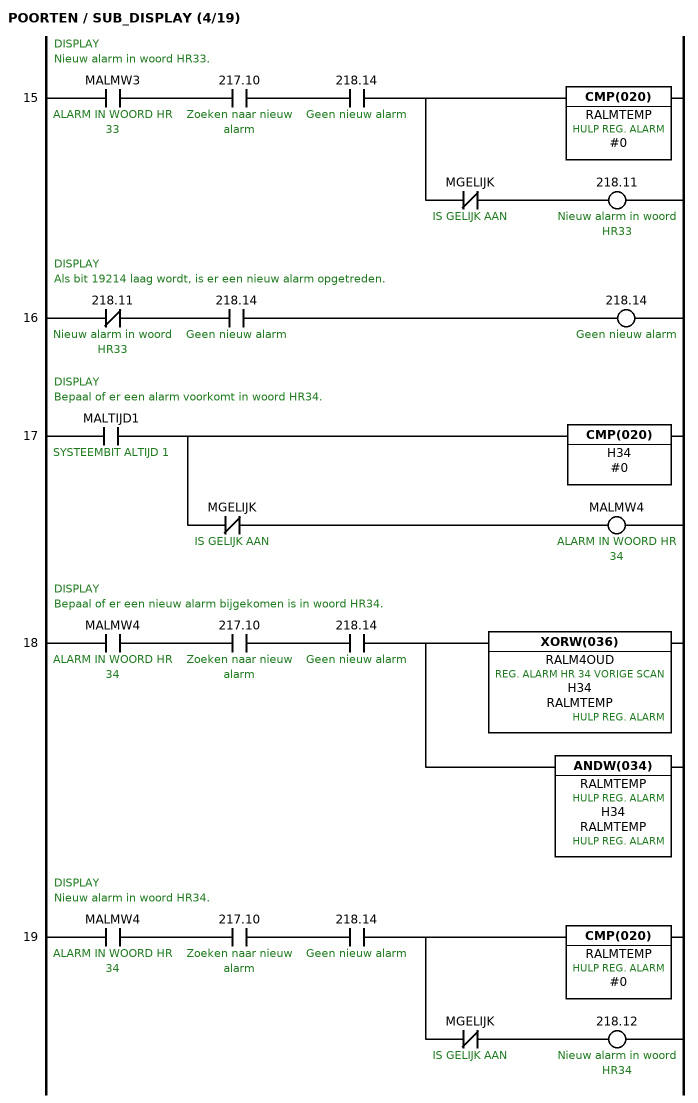
; [picture p469: POORTEN / SUB_DISPLAY, rungs 15-19]
; rung 15: DISPLAY / Nieuw alarm in woord HR33.
LD MALMW3  ; ALARM IN WOORD HR 33
AND 217.10  ; Zoeken naar nieuw alarm
AND 218.14  ; Geen nieuw alarm
CMP(020) RALMTEMP #0  ; HULP REG. ALARM
ANDNOT MGELIJK  ; IS GELIJK AAN
OUT 218.11  ; Nieuw alarm in woord HR33
; rung 16: DISPLAY / Als bit 19214 laag wordt, is er een nieuw alarm opgetreden.
LDNOT 218.11  ; Nieuw alarm in woord HR33
AND 218.14  ; Geen nieuw alarm
OUT 218.14  ; Geen nieuw alarm
; rung 17: DISPLAY / Bepaal of er een alarm voorkomt in woord HR34.
LD MALTIJD1  ; SYSTEEMBIT ALTIJD 1
CMP(020) H34 #0
ANDNOT MGELIJK  ; IS GELIJK AAN
OUT MALMW4  ; ALARM IN WOORD HR 34
; rung 18: DISPLAY / Bepaal of er een nieuw alarm bijgekomen is in woord HR34.
LD MALMW4  ; ALARM IN WOORD HR 34
AND 217.10  ; Zoeken naar nieuw alarm
AND 218.14  ; Geen nieuw alarm
XORW(036) RALM4OUD H34 RALMTEMP  ; REG. ALARM HR 34 VORIGE SCAN, HULP REG. ALARM
ANDW(034) RALMTEMP H34 RALMTEMP  ; HULP REG. ALARM
; rung 19: DISPLAY / Nieuw alarm in woord HR34.
LD MALMW4  ; ALARM IN WOORD HR 34
AND 217.10  ; Zoeken naar nieuw alarm
AND 218.14  ; Geen nieuw alarm
CMP(020) RALMTEMP #0  ; HULP REG. ALARM
ANDNOT MGELIJK  ; IS GELIJK AAN
OUT 218.12  ; Nieuw alarm in woord HR34

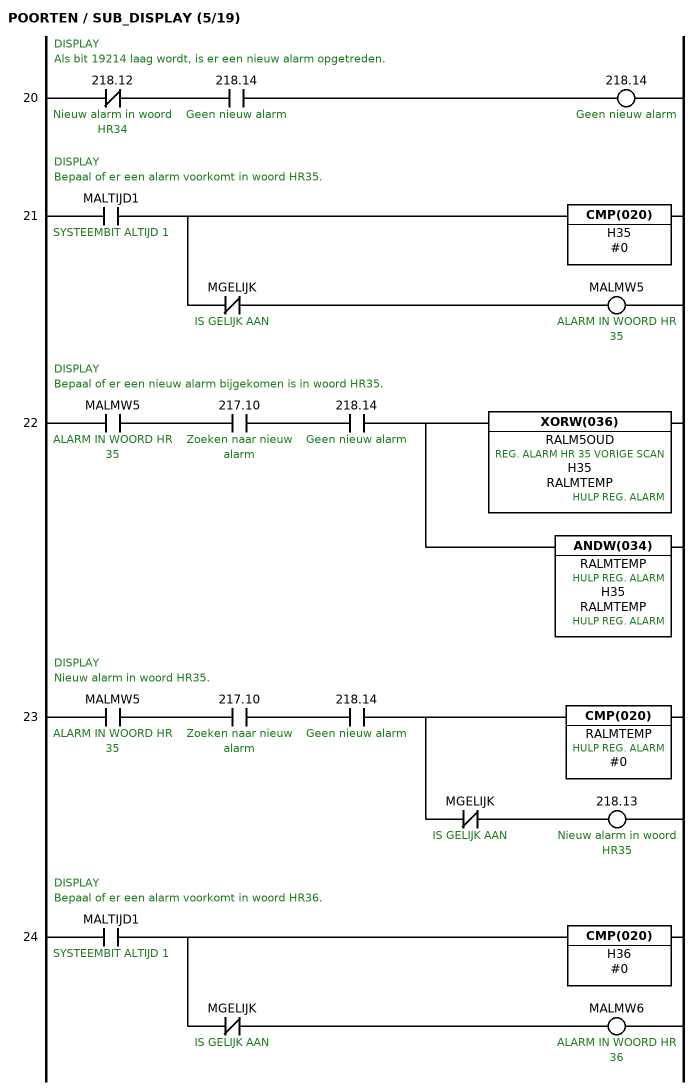
; rung 20: DISPLAY / Als bit 19214 laag wordt, is er een nieuw alarm opgetreden.
LDNOT 218.12  ; Nieuw alarm in woord HR34
AND 218.14  ; Geen nieuw alarm
OUT 218.14  ; Geen nieuw alarm
; rung 21: DISPLAY / Bepaal of er een alarm voorkomt in woord HR35.
LD MALTIJD1  ; SYSTEEMBIT ALTIJD 1
CMP(020) H35 #0
ANDNOT MGELIJK  ; IS GELIJK AAN
OUT MALMW5  ; ALARM IN WOORD HR 35
; rung 22: DISPLAY / Bepaal of er een nieuw alarm bijgekomen is in woord HR35.
LD MALMW5  ; ALARM IN WOORD HR 35
AND 217.10  ; Zoeken naar nieuw alarm
AND 218.14  ; Geen nieuw alarm
XORW(036) RALM5OUD H35 RALMTEMP  ; REG. ALARM HR 35 VORIGE SCAN, HULP REG. ALARM
ANDW(034) RALMTEMP H35 RALMTEMP  ; HULP REG. ALARM
; rung 23: DISPLAY / Nieuw alarm in woord HR35.
LD MALMW5  ; ALARM IN WOORD HR 35
AND 217.10  ; Zoeken naar nieuw alarm
AND 218.14  ; Geen nieuw alarm
CMP(020) RALMTEMP #0  ; HULP REG. ALARM
ANDNOT MGELIJK  ; IS GELIJK AAN
OUT 218.13  ; Nieuw alarm in woord HR35
; rung 24: DISPLAY / Bepaal of er een alarm voorkomt in woord HR36.
LD MALTIJD1  ; SYSTEEMBIT ALTIJD 1
CMP(020) H36 #0
ANDNOT MGELIJK  ; IS GELIJK AAN
OUT MALMW6  ; ALARM IN WOORD HR 36

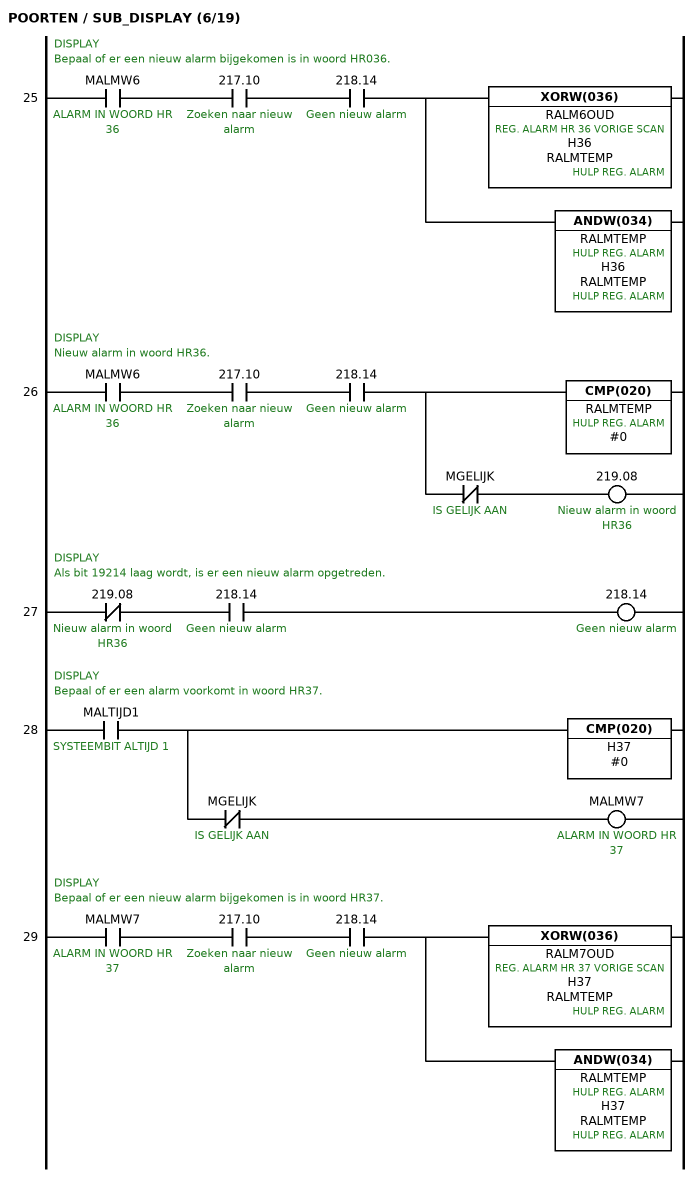
; rung 25: DISPLAY / Bepaal of er een nieuw alarm bijgekomen is in woord HR036.
LD MALMW6  ; ALARM IN WOORD HR 36
AND 217.10  ; Zoeken naar nieuw alarm
AND 218.14  ; Geen nieuw alarm
XORW(036) RALM6OUD H36 RALMTEMP  ; REG. ALARM HR 36 VORIGE SCAN, HULP REG. ALARM
ANDW(034) RALMTEMP H36 RALMTEMP  ; HULP REG. ALARM
; rung 26: DISPLAY / Nieuw alarm in woord HR36.
LD MALMW6  ; ALARM IN WOORD HR 36
AND 217.10  ; Zoeken naar nieuw alarm
AND 218.14  ; Geen nieuw alarm
CMP(020) RALMTEMP #0  ; HULP REG. ALARM
ANDNOT MGELIJK  ; IS GELIJK AAN
OUT 219.08  ; Nieuw alarm in woord HR36
; rung 27: DISPLAY / Als bit 19214 laag wordt, is er een nieuw alarm opgetreden.
LDNOT 219.08  ; Nieuw alarm in woord HR36
AND 218.14  ; Geen nieuw alarm
OUT 218.14  ; Geen nieuw alarm
; rung 28: DISPLAY / Bepaal of er een alarm voorkomt in woord HR37.
LD MALTIJD1  ; SYSTEEMBIT ALTIJD 1
CMP(020) H37 #0
ANDNOT MGELIJK  ; IS GELIJK AAN
OUT MALMW7  ; ALARM IN WOORD HR 37
; rung 29: DISPLAY / Bepaal of er een nieuw alarm bijgekomen is in woord HR37.
LD MALMW7  ; ALARM IN WOORD HR 37
AND 217.10  ; Zoeken naar nieuw alarm
AND 218.14  ; Geen nieuw alarm
XORW(036) RALM7OUD H37 RALMTEMP  ; REG. ALARM HR 37 VORIGE SCAN, HULP REG. ALARM
ANDW(034) RALMTEMP H37 RALMTEMP  ; HULP REG. ALARM

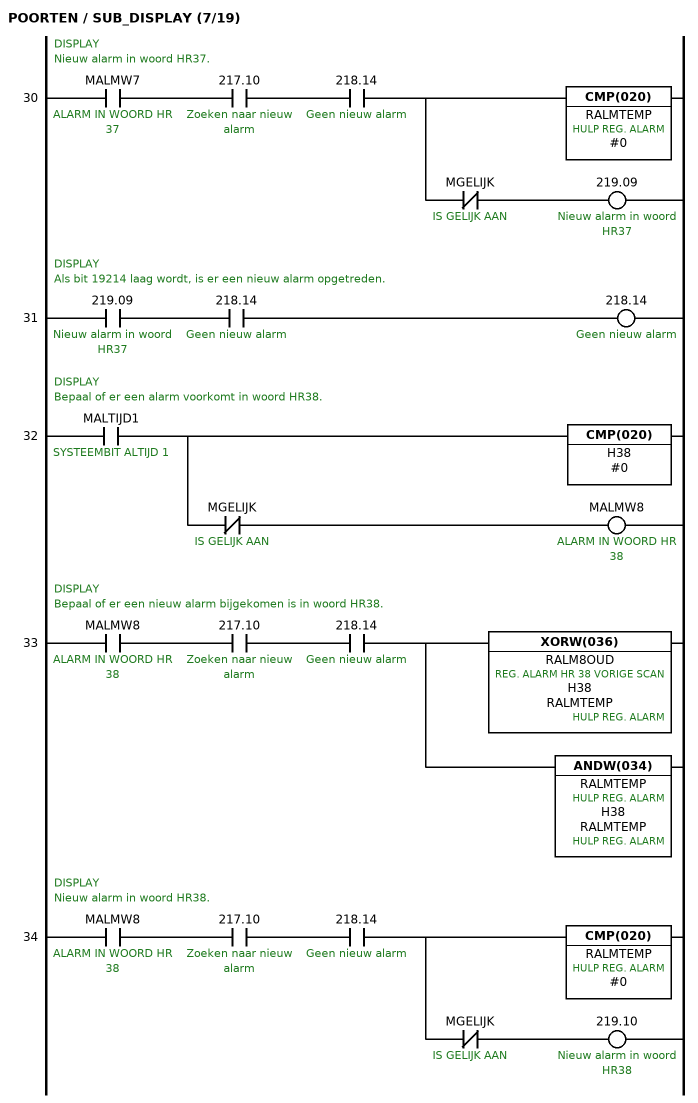
; rung 30: DISPLAY / Nieuw alarm in woord HR37.
LD MALMW7  ; ALARM IN WOORD HR 37
AND 217.10  ; Zoeken naar nieuw alarm
AND 218.14  ; Geen nieuw alarm
CMP(020) RALMTEMP #0  ; HULP REG. ALARM
ANDNOT MGELIJK  ; IS GELIJK AAN
OUT 219.09  ; Nieuw alarm in woord HR37
; rung 31: DISPLAY / Als bit 19214 laag wordt, is er een nieuw alarm opgetreden.
LD 219.09  ; Nieuw alarm in woord HR37
AND 218.14  ; Geen nieuw alarm
OUT 218.14  ; Geen nieuw alarm
; rung 32: DISPLAY / Bepaal of er een alarm voorkomt in woord HR38.
LD MALTIJD1  ; SYSTEEMBIT ALTIJD 1
CMP(020) H38 #0
ANDNOT MGELIJK  ; IS GELIJK AAN
OUT MALMW8  ; ALARM IN WOORD HR 38
; rung 33: DISPLAY / Bepaal of er een nieuw alarm bijgekomen is in woord HR38.
LD MALMW8  ; ALARM IN WOORD HR 38
AND 217.10  ; Zoeken naar nieuw alarm
AND 218.14  ; Geen nieuw alarm
XORW(036) RALM8OUD H38 RALMTEMP  ; REG. ALARM HR 38 VORIGE SCAN, HULP REG. ALARM
ANDW(034) RALMTEMP H38 RALMTEMP  ; HULP REG. ALARM
; rung 34: DISPLAY / Nieuw alarm in woord HR38.
LD MALMW8  ; ALARM IN WOORD HR 38
AND 217.10  ; Zoeken naar nieuw alarm
AND 218.14  ; Geen nieuw alarm
CMP(020) RALMTEMP #0  ; HULP REG. ALARM
ANDNOT MGELIJK  ; IS GELIJK AAN
OUT 219.10  ; Nieuw alarm in woord HR38

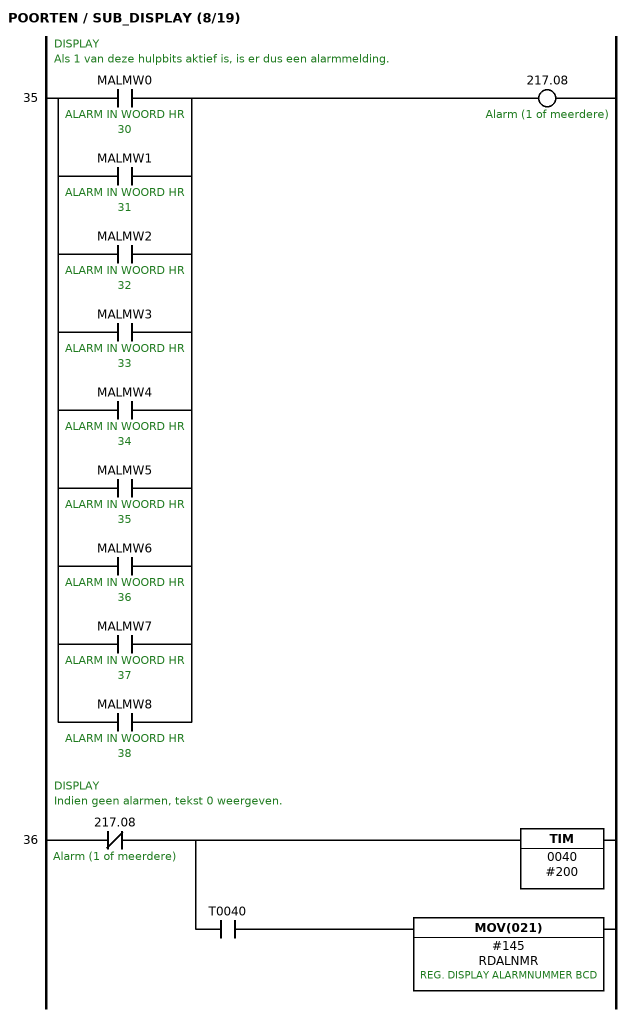
; rung 35: DISPLAY / Als 1 van deze hulpbits aktief is, is er dus een alarmmelding.
LD MALMW0  ; ALARM IN WOORD HR 30
OR MALMW1  ; ALARM IN WOORD HR 31
OR MALMW2  ; ALARM IN WOORD HR 32
OR MALMW3  ; ALARM IN WOORD HR 33
OR MALMW4  ; ALARM IN WOORD HR 34
OR MALMW5  ; ALARM IN WOORD HR 35
OR MALMW6  ; ALARM IN WOORD HR 36
OR MALMW7  ; ALARM IN WOORD HR 37
OR MALMW8  ; ALARM IN WOORD HR 38
OUT 217.08  ; Alarm (1 of meerdere)
; rung 36: DISPLAY / Indien geen alarmen, tekst 0 weergeven.
LDNOT 217.08  ; Alarm (1 of meerdere)
TIM 0040 #200
AND T0040
MOV(021) #145 RDALNMR  ; REG. DISPLAY ALARMNUMMER BCD

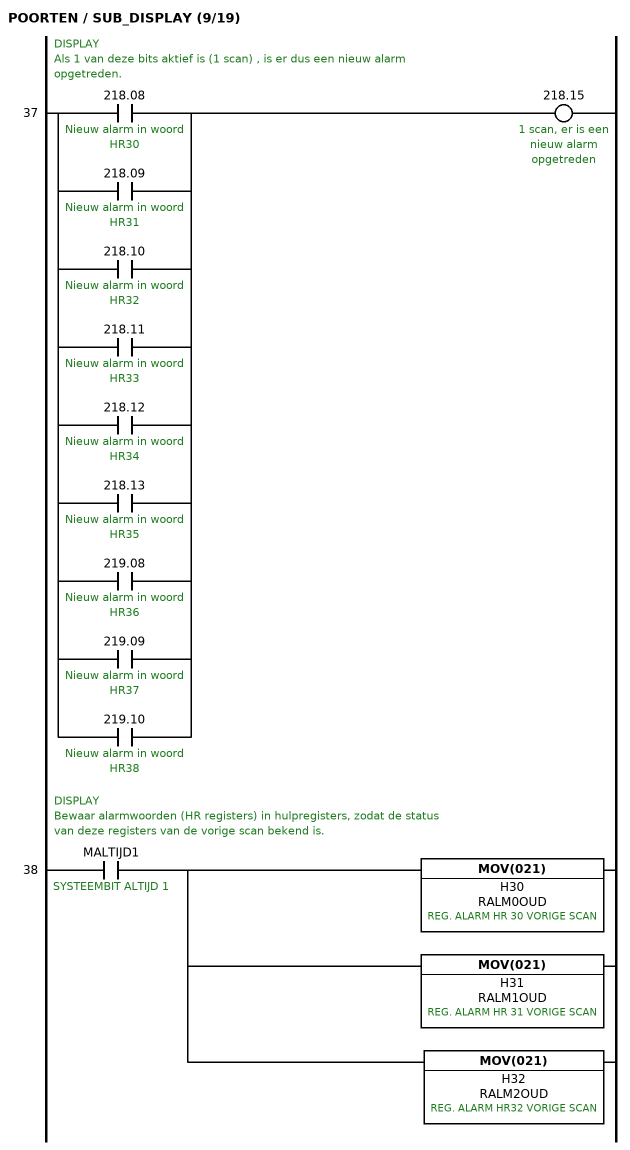
; rung 37: DISPLAY / Als 1 van deze bits aktief is (1 scan) , is er dus een nieuw alarm / opgetreden.
LD 218.08  ; Nieuw alarm in woord HR30
OR 218.09  ; Nieuw alarm in woord HR31
OR 218.10  ; Nieuw alarm in woord HR32
OR 218.11  ; Nieuw alarm in woord HR33
OR 218.12  ; Nieuw alarm in woord HR34
OR 218.13  ; Nieuw alarm in woord HR35
OR 219.08  ; Nieuw alarm in woord HR36
OR 219.09  ; Nieuw alarm in woord HR37
OR 219.10  ; Nieuw alarm in woord HR38
OUT 218.15  ; 1 scan, er is een nieuw alarm opgetreden
; rung 38: DISPLAY / Bewaar alarmwoorden (HR registers) in hulpregisters, zodat de status / van deze registers van de vorige scan bekend is.
LD MALTIJD1  ; SYSTEEMBIT ALTIJD 1
MOV(021) H30 RALM0OUD  ; REG. ALARM HR 30 VORIGE SCAN
MOV(021) H31 RALM1OUD  ; REG. ALARM HR 31 VORIGE SCAN
MOV(021) H32 RALM2OUD  ; REG. ALARM HR32 VORIGE SCAN

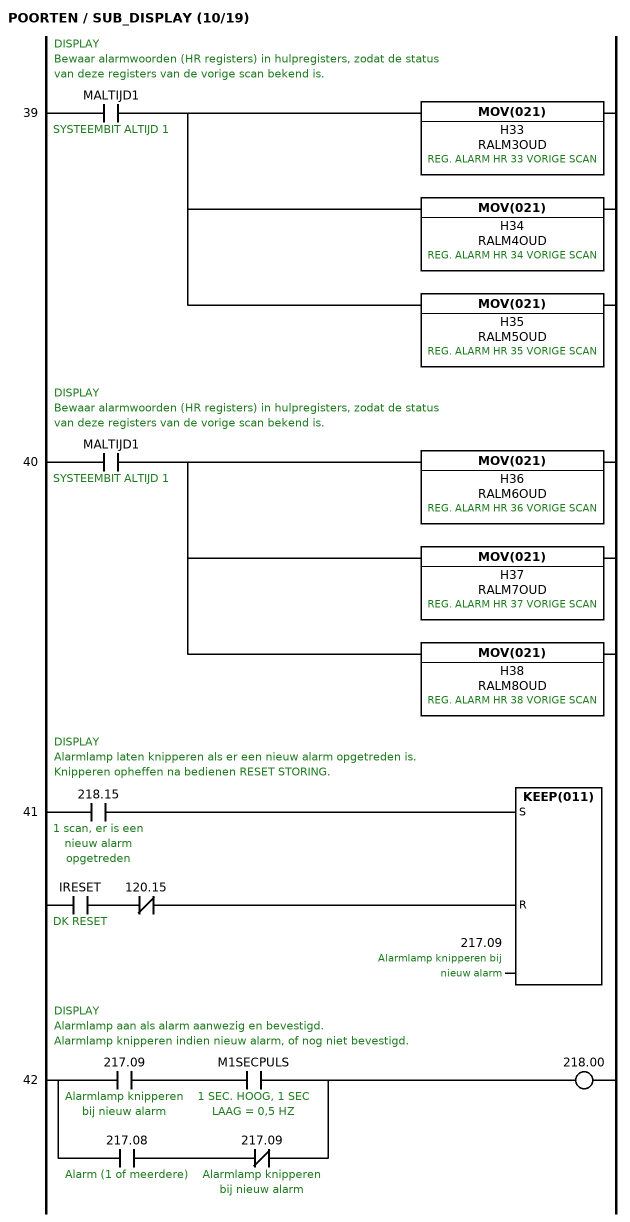
; rung 39: DISPLAY / Bewaar alarmwoorden (HR registers) in hulpregisters, zodat de status / van deze registers van de vorige scan bekend is.
LD MALTIJD1  ; SYSTEEMBIT ALTIJD 1
MOV(021) H33 RALM3OUD  ; REG. ALARM HR 33 VORIGE SCAN
MOV(021) H34 RALM4OUD  ; REG. ALARM HR 34 VORIGE SCAN
MOV(021) H35 RALM5OUD  ; REG. ALARM HR 35 VORIGE SCAN
; rung 40: DISPLAY / Bewaar alarmwoorden (HR registers) in hulpregisters, zodat de status / van deze registers van de vorige scan bekend is.
LD MALTIJD1  ; SYSTEEMBIT ALTIJD 1
MOV(021) H36 RALM6OUD  ; REG. ALARM HR 36 VORIGE SCAN
MOV(021) H37 RALM7OUD  ; REG. ALARM HR 37 VORIGE SCAN
MOV(021) H38 RALM8OUD  ; REG. ALARM HR 38 VORIGE SCAN
; rung 41: DISPLAY / Alarmlamp laten knipperen als er een nieuw alarm opgetreden is. / Knipperen opheffen na bedienen RESET STORING.
LD 218.15  ; 1 scan, er is een nieuw alarm opgetreden
LD IRESET  ; DK RESET
ANDNOT 120.15
KEEP(011) 217.09  ; Alarmlamp knipperen bij nieuw alarm
; rung 42: DISPLAY / Alarmlamp aan als alarm aanwezig en bevestigd. / Alarmlamp knipperen indien nieuw alarm, of nog niet bevestigd.
LD 217.09  ; Alarmlamp knipperen bij nieuw alarm
AND M1SECPULS  ; 1 SEC. HOOG, 1 SEC LAAG = 0,5 HZ
LD 217.08  ; Alarm (1 of meerdere)
ANDNOT 217.09  ; Alarmlamp knipperen bij nieuw alarm
ORLD
OUT 218.00

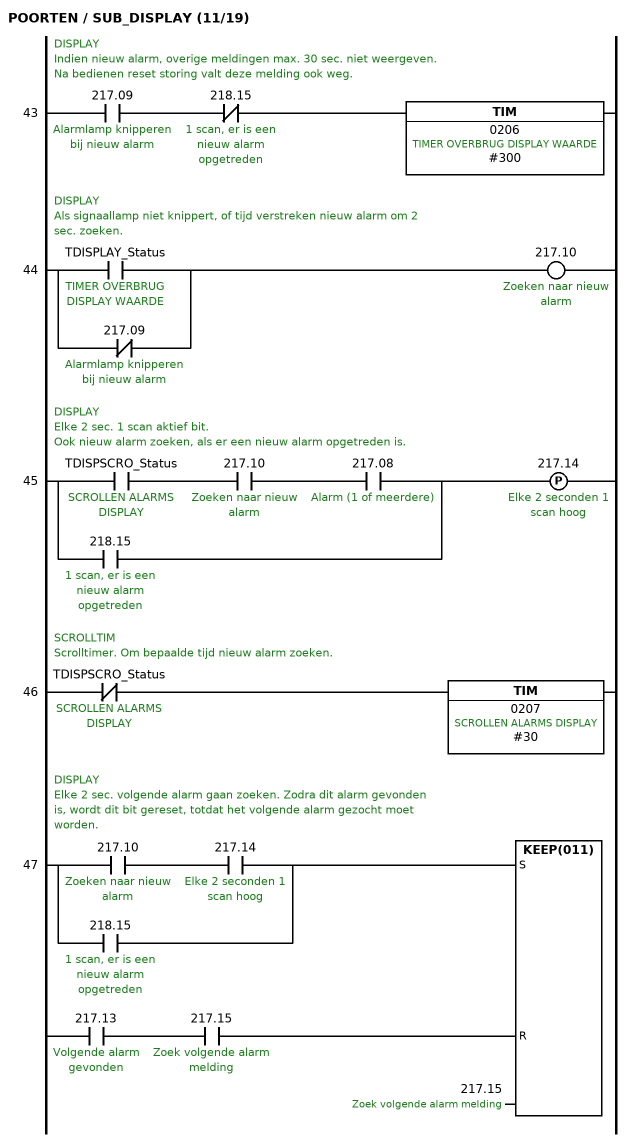
; rung 43: DISPLAY / Indien nieuw alarm, overige meldingen max. 30 sec. niet weergeven. / Na bedienen reset storing valt deze melding ook weg.
LD 217.09  ; Alarmlamp knipperen bij nieuw alarm
ANDNOT 218.15  ; 1 scan, er is een nieuw alarm opgetreden
TIM 0206 #300  ; TIMER OVERBRUG DISPLAY WAARDE
; rung 44: DISPLAY / Als signaallamp niet knippert, of tijd verstreken nieuw alarm om 2 / sec. zoeken.
LD TDISPLAY_Status  ; TIMER OVERBRUG DISPLAY WAARDE
ORNOT 217.09  ; Alarmlamp knipperen bij nieuw alarm
OUT 217.10  ; Zoeken naar nieuw alarm
; rung 45: DISPLAY / Elke 2 sec. 1 scan aktief bit. / Ook nieuw alarm zoeken, als er een nieuw alarm opgetreden is.
LD TDISPSCRO_Status  ; SCROLLEN ALARMS DISPLAY
AND 217.10  ; Zoeken naar nieuw alarm
AND 217.08  ; Alarm (1 of meerdere)
OR 218.15  ; 1 scan, er is een nieuw alarm opgetreden
DIFU(013) 217.14  ; Elke 2 seconden 1 scan hoog
; rung 46: SCROLLTIM / Scrolltimer. Om bepaalde tijd nieuw alarm zoeken.
LDNOT TDISPSCRO_Status  ; SCROLLEN ALARMS DISPLAY
TIM 0207 #30  ; SCROLLEN ALARMS DISPLAY
; rung 47: DISPLAY / Elke 2 sec. volgende alarm gaan zoeken. Zodra dit alarm gevonden / is, wordt dit bit gereset, totdat het volgende alarm gezocht moet / worden.
LD 217.10  ; Zoeken naar nieuw alarm
AND 217.14  ; Elke 2 seconden 1 scan hoog
OR 218.15  ; 1 scan, er is een nieuw alarm opgetreden
LD 217.13  ; Volgende alarm gevonden
AND 217.15  ; Zoek volgende alarm melding
KEEP(011) 217.15  ; Zoek volgende alarm melding

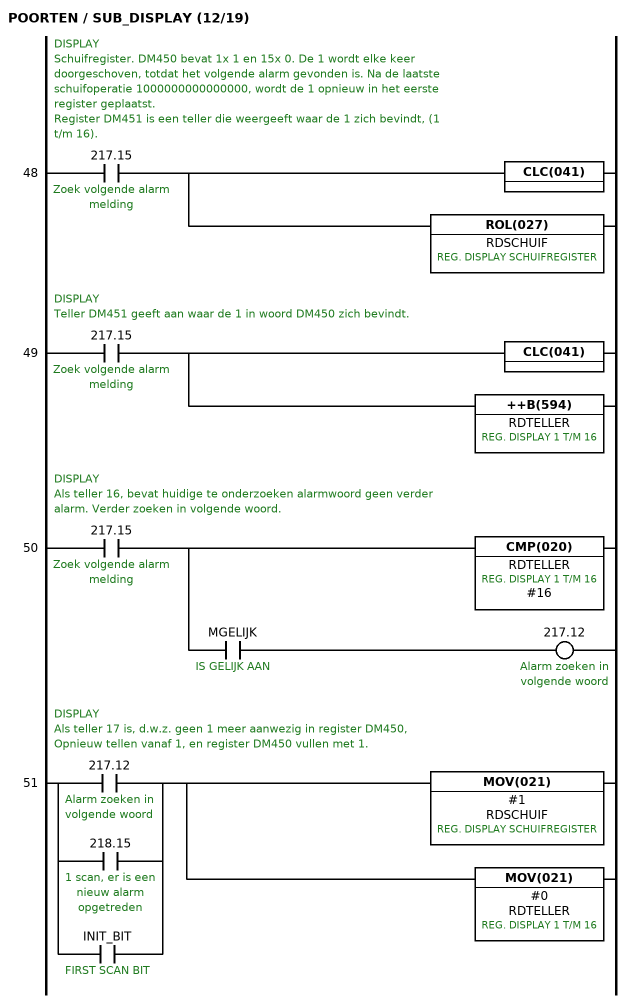
; rung 48: DISPLAY / Schuifregister. DM450 bevat 1x 1 en 15x 0. De 1 wordt elke keer / doorgeschoven, totdat het volgende alarm gevonden is. Na de laatste / schuifoperatie 1000000000000000, wordt de 1 opnieuw in het eerste / register geplaatst. / Register DM451 is een teller die weergeeft waar de 1 zich bevindt, (1 / t/m 16).
LD 217.15  ; Zoek volgende alarm melding
CLC(041)
ROL(027) RDSCHUIF  ; REG. DISPLAY SCHUIFREGISTER
; rung 49: DISPLAY / Teller DM451 geeft aan waar de 1 in woord DM450 zich bevindt.
LD 217.15  ; Zoek volgende alarm melding
CLC(041)
++B(594) RDTELLER  ; REG. DISPLAY 1 T/M 16
; rung 50: DISPLAY / Als teller 16, bevat huidige te onderzoeken alarmwoord geen verder / alarm. Verder zoeken in volgende woord.
LD 217.15  ; Zoek volgende alarm melding
CMP(020) RDTELLER #16  ; REG. DISPLAY 1 T/M 16
AND MGELIJK  ; IS GELIJK AAN
OUT 217.12  ; Alarm zoeken in volgende woord
; rung 51: DISPLAY / Als teller 17 is, d.w.z. geen 1 meer aanwezig in register DM450, / Opnieuw tellen vanaf 1, en register DM450 vullen met 1.
LD 217.12  ; Alarm zoeken in volgende woord
OR 218.15  ; 1 scan, er is een nieuw alarm opgetreden
OR INIT_BIT  ; FIRST SCAN BIT
MOV(021) #1 RDSCHUIF  ; REG. DISPLAY SCHUIFREGISTER
MOV(021) #0 RDTELLER  ; REG. DISPLAY 1 T/M 16

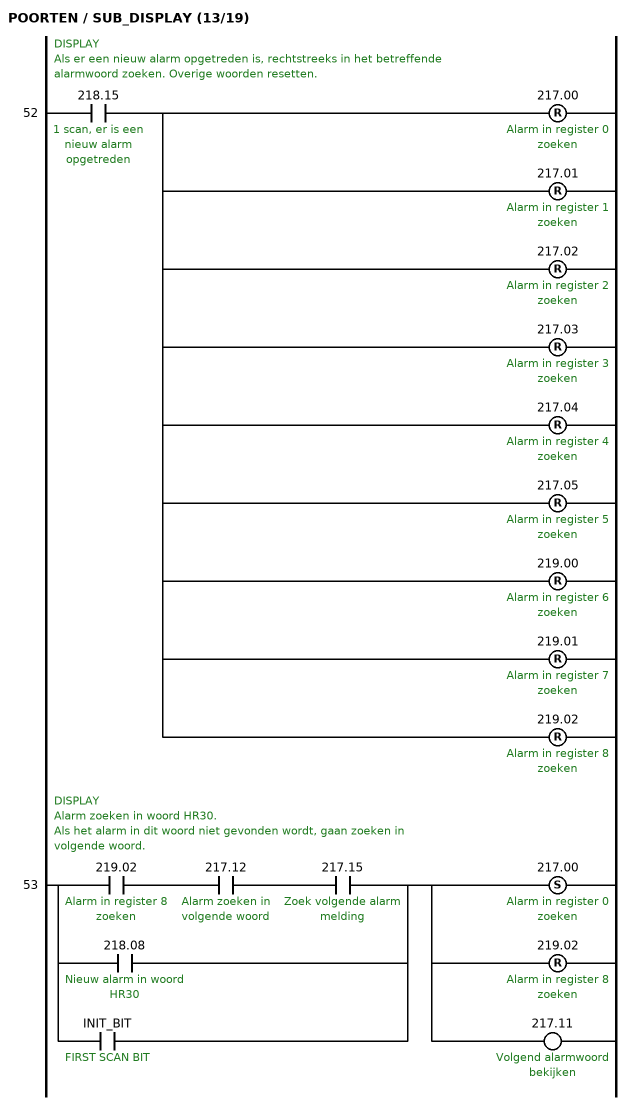
; rung 52: DISPLAY / Als er een nieuw alarm opgetreden is, rechtstreeks in het betreffende / alarmwoord zoeken. Overige woorden resetten.
LD 218.15  ; 1 scan, er is een nieuw alarm opgetreden
RSET 217.00  ; Alarm in register 0 zoeken
RSET 217.01  ; Alarm in register 1 zoeken
RSET 217.02  ; Alarm in register 2 zoeken
RSET 217.03  ; Alarm in register 3 zoeken
RSET 217.04  ; Alarm in register 4 zoeken
RSET 217.05  ; Alarm in register 5 zoeken
RSET 219.00  ; Alarm in register 6 zoeken
RSET 219.01  ; Alarm in register 7 zoeken
RSET 219.02  ; Alarm in register 8 zoeken
; rung 53: DISPLAY / Alarm zoeken in woord HR30. / Als het alarm in dit woord niet gevonden wordt, gaan zoeken in / volgende woord.
LD 219.02  ; Alarm in register 8 zoeken
AND 217.12  ; Alarm zoeken in volgende woord
AND 217.15  ; Zoek volgende alarm melding
OR 218.08  ; Nieuw alarm in woord HR30
OR INIT_BIT  ; FIRST SCAN BIT
SET 217.00  ; Alarm in register 0 zoeken
RSET 219.02  ; Alarm in register 8 zoeken
OUT 217.11  ; Volgend alarmwoord bekijken

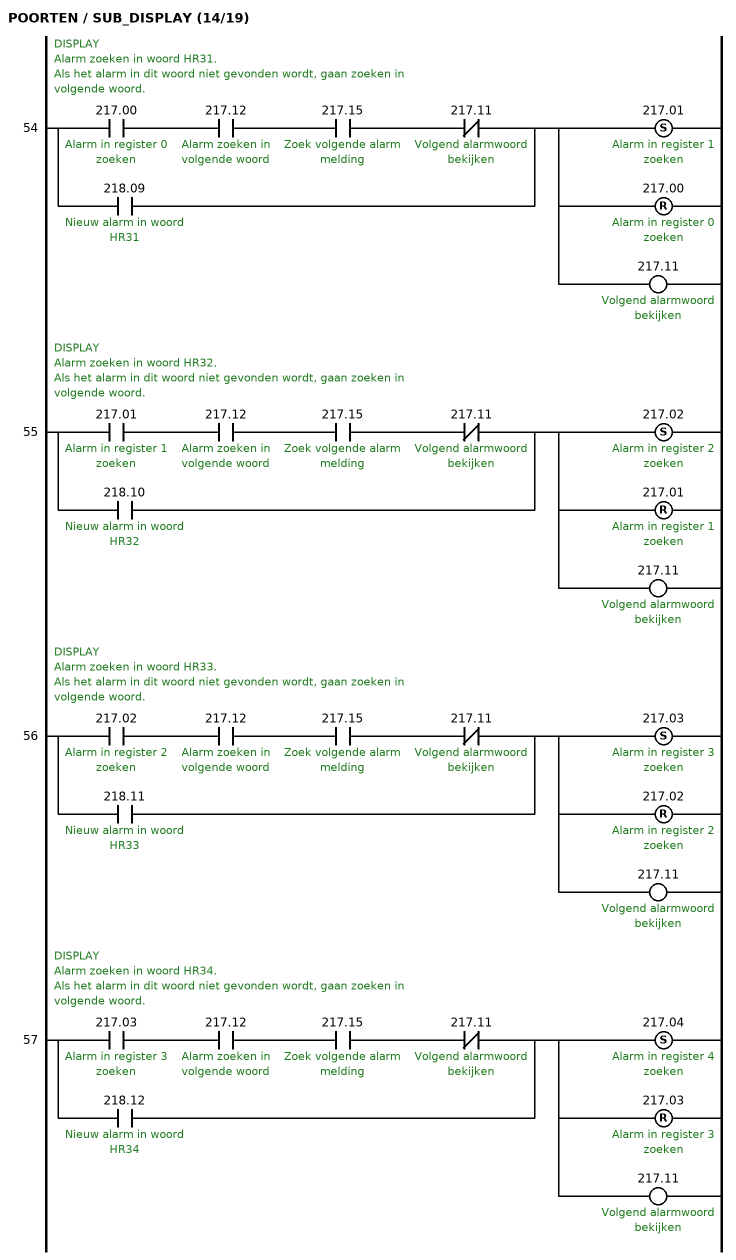
; rung 54: DISPLAY / Alarm zoeken in woord HR31. / Als het alarm in dit woord niet gevonden wordt, gaan zoeken in / volgende woord.
LD 217.00  ; Alarm in register 0 zoeken
AND 217.12  ; Alarm zoeken in volgende woord
AND 217.15  ; Zoek volgende alarm melding
ANDNOT 217.11  ; Volgend alarmwoord bekijken
OR 218.09  ; Nieuw alarm in woord HR31
SET 217.01  ; Alarm in register 1 zoeken
RSET 217.00  ; Alarm in register 0 zoeken
OUT 217.11  ; Volgend alarmwoord bekijken
; rung 55: DISPLAY / Alarm zoeken in woord HR32. / Als het alarm in dit woord niet gevonden wordt, gaan zoeken in / volgende woord.
LD 217.01  ; Alarm in register 1 zoeken
AND 217.12  ; Alarm zoeken in volgende woord
AND 217.15  ; Zoek volgende alarm melding
ANDNOT 217.11  ; Volgend alarmwoord bekijken
OR 218.10  ; Nieuw alarm in woord HR32
SET 217.02  ; Alarm in register 2 zoeken
RSET 217.01  ; Alarm in register 1 zoeken
OUT 217.11  ; Volgend alarmwoord bekijken
; rung 56: DISPLAY / Alarm zoeken in woord HR33. / Als het alarm in dit woord niet gevonden wordt, gaan zoeken in / volgende woord.
LD 217.02  ; Alarm in register 2 zoeken
AND 217.12  ; Alarm zoeken in volgende woord
AND 217.15  ; Zoek volgende alarm melding
ANDNOT 217.11  ; Volgend alarmwoord bekijken
OR 218.11  ; Nieuw alarm in woord HR33
SET 217.03  ; Alarm in register 3 zoeken
RSET 217.02  ; Alarm in register 2 zoeken
OUT 217.11  ; Volgend alarmwoord bekijken
; rung 57: DISPLAY / Alarm zoeken in woord HR34. / Als het alarm in dit woord niet gevonden wordt, gaan zoeken in / volgende woord.
LD 217.03  ; Alarm in register 3 zoeken
AND 217.12  ; Alarm zoeken in volgende woord
AND 217.15  ; Zoek volgende alarm melding
ANDNOT 217.11  ; Volgend alarmwoord bekijken
OR 218.12  ; Nieuw alarm in woord HR34
SET 217.04  ; Alarm in register 4 zoeken
RSET 217.03  ; Alarm in register 3 zoeken
OUT 217.11  ; Volgend alarmwoord bekijken

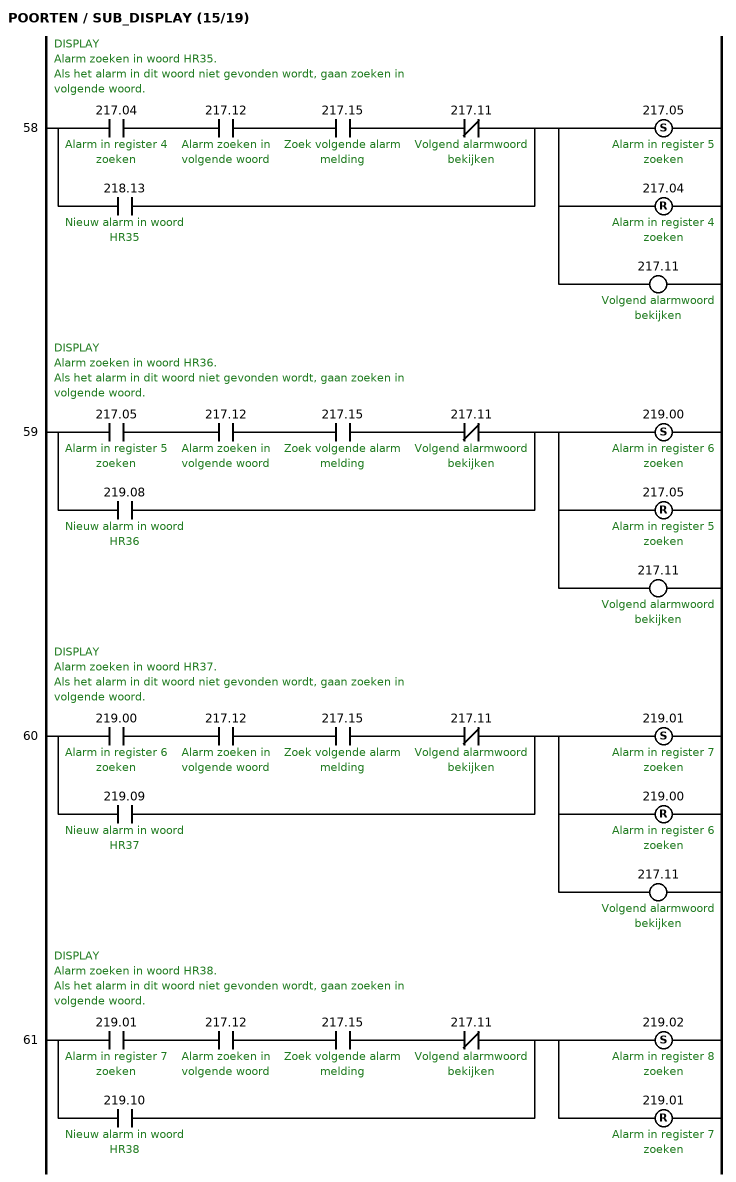
; rung 58: DISPLAY / Alarm zoeken in woord HR35. / Als het alarm in dit woord niet gevonden wordt, gaan zoeken in / volgende woord.
LD 217.04  ; Alarm in register 4 zoeken
AND 217.12  ; Alarm zoeken in volgende woord
AND 217.15  ; Zoek volgende alarm melding
ANDNOT 217.11  ; Volgend alarmwoord bekijken
OR 218.13  ; Nieuw alarm in woord HR35
SET 217.05  ; Alarm in register 5 zoeken
RSET 217.04  ; Alarm in register 4 zoeken
OUT 217.11  ; Volgend alarmwoord bekijken
; rung 59: DISPLAY / Alarm zoeken in woord HR36. / Als het alarm in dit woord niet gevonden wordt, gaan zoeken in / volgende woord.
LD 217.05  ; Alarm in register 5 zoeken
AND 217.12  ; Alarm zoeken in volgende woord
AND 217.15  ; Zoek volgende alarm melding
ANDNOT 217.11  ; Volgend alarmwoord bekijken
OR 219.08  ; Nieuw alarm in woord HR36
SET 219.00  ; Alarm in register 6 zoeken
RSET 217.05  ; Alarm in register 5 zoeken
OUT 217.11  ; Volgend alarmwoord bekijken
; rung 60: DISPLAY / Alarm zoeken in woord HR37. / Als het alarm in dit woord niet gevonden wordt, gaan zoeken in / volgende woord.
LD 219.00  ; Alarm in register 6 zoeken
AND 217.12  ; Alarm zoeken in volgende woord
AND 217.15  ; Zoek volgende alarm melding
ANDNOT 217.11  ; Volgend alarmwoord bekijken
OR 219.09  ; Nieuw alarm in woord HR37
SET 219.01  ; Alarm in register 7 zoeken
RSET 219.00  ; Alarm in register 6 zoeken
OUT 217.11  ; Volgend alarmwoord bekijken
; rung 61: DISPLAY / Alarm zoeken in woord HR38. / Als het alarm in dit woord niet gevonden wordt, gaan zoeken in / volgende woord.
LD 219.01  ; Alarm in register 7 zoeken
AND 217.12  ; Alarm zoeken in volgende woord
AND 217.15  ; Zoek volgende alarm melding
ANDNOT 217.11  ; Volgend alarmwoord bekijken
OR 219.10  ; Nieuw alarm in woord HR38
SET 219.02  ; Alarm in register 8 zoeken
RSET 219.01  ; Alarm in register 7 zoeken

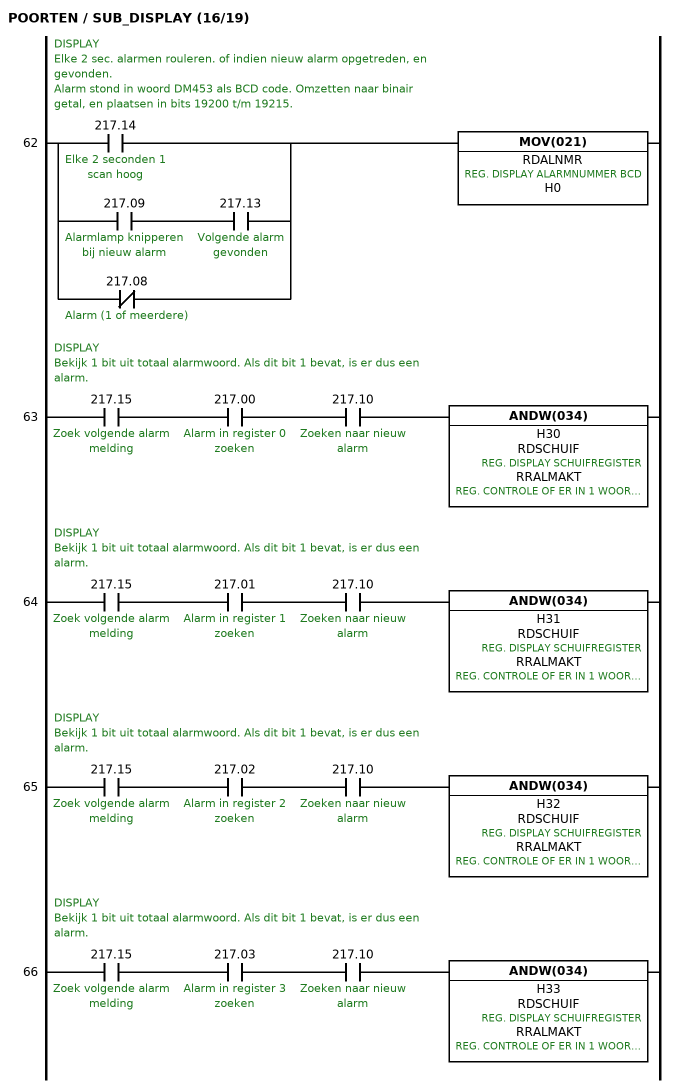
; rung 62: DISPLAY / Elke 2 sec. alarmen rouleren. of indien nieuw alarm opgetreden, en / gevonden. / Alarm stond in woord DM453 als BCD code. Omzetten naar binair / getal, en plaatsen in bits 19200 t/m 19215.
LD 217.14  ; Elke 2 seconden 1 scan hoog
LD 217.09  ; Alarmlamp knipperen bij nieuw alarm
AND 217.13  ; Volgende alarm gevonden
ORLD
ORNOT 217.08  ; Alarm (1 of meerdere)
MOV(021) RDALNMR H0  ; REG. DISPLAY ALARMNUMMER BCD
; rung 63: DISPLAY / Bekijk 1 bit uit totaal alarmwoord. Als dit bit 1 bevat, is er dus een / alarm.
LD 217.15  ; Zoek volgende alarm melding
AND 217.00  ; Alarm in register 0 zoeken
AND 217.10  ; Zoeken naar nieuw alarm
ANDW(034) H30 RDSCHUIF RRALMAKT  ; REG. DISPLAY SCHUIFREGISTER, REG. CONTROLE OF ER IN 1 WOORD EEN ALARM HOOG IS
; rung 64: DISPLAY / Bekijk 1 bit uit totaal alarmwoord. Als dit bit 1 bevat, is er dus een / alarm.
LD 217.15  ; Zoek volgende alarm melding
AND 217.01  ; Alarm in register 1 zoeken
AND 217.10  ; Zoeken naar nieuw alarm
ANDW(034) H31 RDSCHUIF RRALMAKT  ; REG. DISPLAY SCHUIFREGISTER, REG. CONTROLE OF ER IN 1 WOORD EEN ALARM HOOG IS
; rung 65: DISPLAY / Bekijk 1 bit uit totaal alarmwoord. Als dit bit 1 bevat, is er dus een / alarm.
LD 217.15  ; Zoek volgende alarm melding
AND 217.02  ; Alarm in register 2 zoeken
AND 217.10  ; Zoeken naar nieuw alarm
ANDW(034) H32 RDSCHUIF RRALMAKT  ; REG. DISPLAY SCHUIFREGISTER, REG. CONTROLE OF ER IN 1 WOORD EEN ALARM HOOG IS
; rung 66: DISPLAY / Bekijk 1 bit uit totaal alarmwoord. Als dit bit 1 bevat, is er dus een / alarm.
LD 217.15  ; Zoek volgende alarm melding
AND 217.03  ; Alarm in register 3 zoeken
AND 217.10  ; Zoeken naar nieuw alarm
ANDW(034) H33 RDSCHUIF RRALMAKT  ; REG. DISPLAY SCHUIFREGISTER, REG. CONTROLE OF ER IN 1 WOORD EEN ALARM HOOG IS

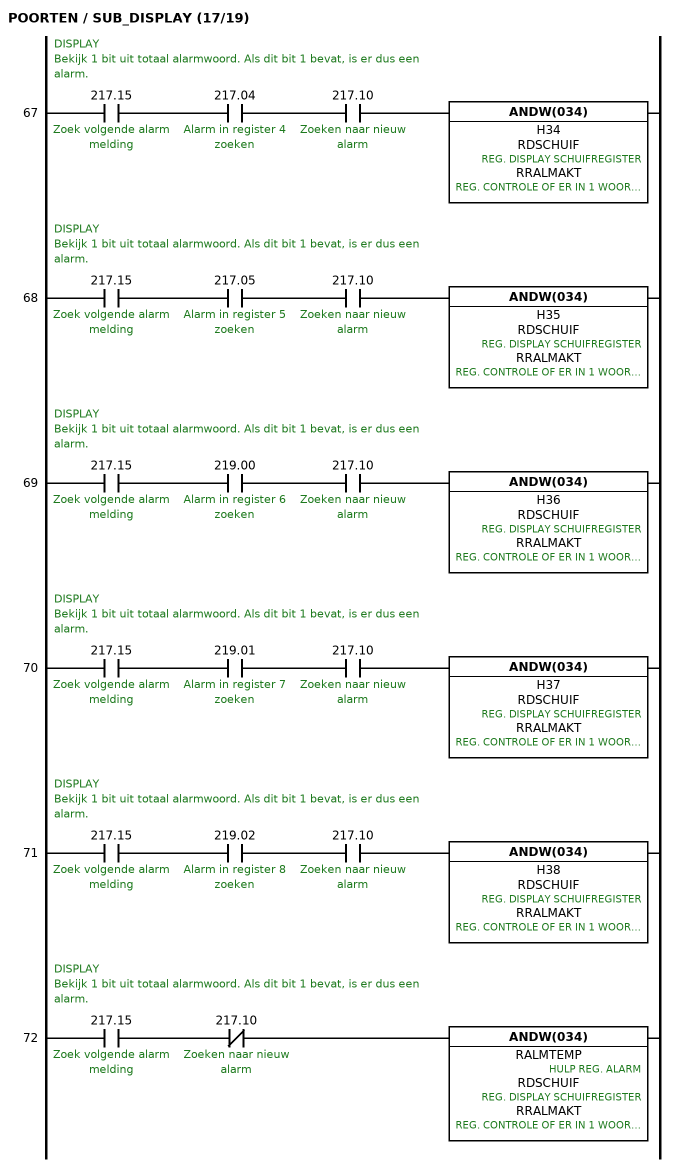
; rung 67: DISPLAY / Bekijk 1 bit uit totaal alarmwoord. Als dit bit 1 bevat, is er dus een / alarm.
LD 217.15  ; Zoek volgende alarm melding
AND 217.04  ; Alarm in register 4 zoeken
AND 217.10  ; Zoeken naar nieuw alarm
ANDW(034) H34 RDSCHUIF RRALMAKT  ; REG. DISPLAY SCHUIFREGISTER, REG. CONTROLE OF ER IN 1 WOORD EEN ALARM HOOG IS
; rung 68: DISPLAY / Bekijk 1 bit uit totaal alarmwoord. Als dit bit 1 bevat, is er dus een / alarm.
LD 217.15  ; Zoek volgende alarm melding
AND 217.05  ; Alarm in register 5 zoeken
AND 217.10  ; Zoeken naar nieuw alarm
ANDW(034) H35 RDSCHUIF RRALMAKT  ; REG. DISPLAY SCHUIFREGISTER, REG. CONTROLE OF ER IN 1 WOORD EEN ALARM HOOG IS
; rung 69: DISPLAY / Bekijk 1 bit uit totaal alarmwoord. Als dit bit 1 bevat, is er dus een / alarm.
LD 217.15  ; Zoek volgende alarm melding
AND 219.00  ; Alarm in register 6 zoeken
AND 217.10  ; Zoeken naar nieuw alarm
ANDW(034) H36 RDSCHUIF RRALMAKT  ; REG. DISPLAY SCHUIFREGISTER, REG. CONTROLE OF ER IN 1 WOORD EEN ALARM HOOG IS
; rung 70: DISPLAY / Bekijk 1 bit uit totaal alarmwoord. Als dit bit 1 bevat, is er dus een / alarm.
LD 217.15  ; Zoek volgende alarm melding
AND 219.01  ; Alarm in register 7 zoeken
AND 217.10  ; Zoeken naar nieuw alarm
ANDW(034) H37 RDSCHUIF RRALMAKT  ; REG. DISPLAY SCHUIFREGISTER, REG. CONTROLE OF ER IN 1 WOORD EEN ALARM HOOG IS
; rung 71: DISPLAY / Bekijk 1 bit uit totaal alarmwoord. Als dit bit 1 bevat, is er dus een / alarm.
LD 217.15  ; Zoek volgende alarm melding
AND 219.02  ; Alarm in register 8 zoeken
AND 217.10  ; Zoeken naar nieuw alarm
ANDW(034) H38 RDSCHUIF RRALMAKT  ; REG. DISPLAY SCHUIFREGISTER, REG. CONTROLE OF ER IN 1 WOORD EEN ALARM HOOG IS
; rung 72: DISPLAY / Bekijk 1 bit uit totaal alarmwoord. Als dit bit 1 bevat, is er dus een / alarm.
LD 217.15  ; Zoek volgende alarm melding
ANDNOT 217.10  ; Zoeken naar nieuw alarm
ANDW(034) RALMTEMP RDSCHUIF RRALMAKT  ; HULP REG. ALARM, REG. DISPLAY SCHUIFREGISTER, REG. CONTROLE OF ER IN 1 WOORD EEN ALARM HOOG IS

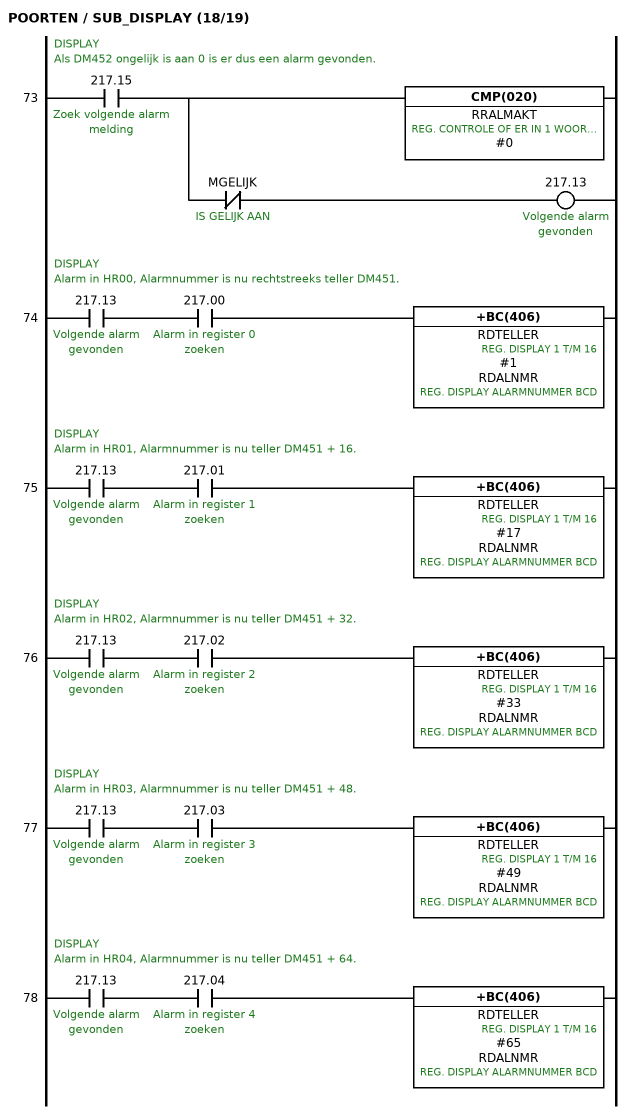
; rung 73: DISPLAY / Als DM452 ongelijk is aan 0 is er dus een alarm gevonden.
LD 217.15  ; Zoek volgende alarm melding
CMP(020) RRALMAKT #0  ; REG. CONTROLE OF ER IN 1 WOORD EEN ALARM HOOG IS
ANDNOT MGELIJK  ; IS GELIJK AAN
OUT 217.13  ; Volgende alarm gevonden
; rung 74: DISPLAY / Alarm in HR00, Alarmnummer is nu rechtstreeks teller DM451.
LD 217.13  ; Volgende alarm gevonden
AND 217.00  ; Alarm in register 0 zoeken
+BC(406) RDTELLER #1 RDALNMR  ; REG. DISPLAY 1 T/M 16, REG. DISPLAY ALARMNUMMER BCD
; rung 75: DISPLAY / Alarm in HR01, Alarmnummer is nu teller DM451 + 16.
LD 217.13  ; Volgende alarm gevonden
AND 217.01  ; Alarm in register 1 zoeken
+BC(406) RDTELLER #17 RDALNMR  ; REG. DISPLAY 1 T/M 16, REG. DISPLAY ALARMNUMMER BCD
; rung 76: DISPLAY / Alarm in HR02, Alarmnummer is nu teller DM451 + 32.
LD 217.13  ; Volgende alarm gevonden
AND 217.02  ; Alarm in register 2 zoeken
+BC(406) RDTELLER #33 RDALNMR  ; REG. DISPLAY 1 T/M 16, REG. DISPLAY ALARMNUMMER BCD
; rung 77: DISPLAY / Alarm in HR03, Alarmnummer is nu teller DM451 + 48.
LD 217.13  ; Volgende alarm gevonden
AND 217.03  ; Alarm in register 3 zoeken
+BC(406) RDTELLER #49 RDALNMR  ; REG. DISPLAY 1 T/M 16, REG. DISPLAY ALARMNUMMER BCD
; rung 78: DISPLAY / Alarm in HR04, Alarmnummer is nu teller DM451 + 64.
LD 217.13  ; Volgende alarm gevonden
AND 217.04  ; Alarm in register 4 zoeken
+BC(406) RDTELLER #65 RDALNMR  ; REG. DISPLAY 1 T/M 16, REG. DISPLAY ALARMNUMMER BCD

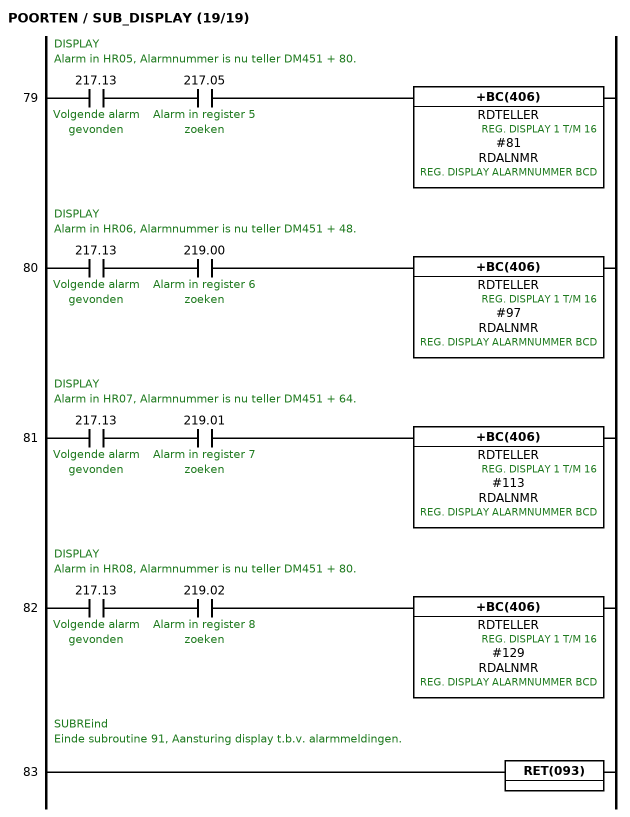
; rung 79: DISPLAY / Alarm in HR05, Alarmnummer is nu teller DM451 + 80.
LD 217.13  ; Volgende alarm gevonden
AND 217.05  ; Alarm in register 5 zoeken
+BC(406) RDTELLER #81 RDALNMR  ; REG. DISPLAY 1 T/M 16, REG. DISPLAY ALARMNUMMER BCD
; rung 80: DISPLAY / Alarm in HR06, Alarmnummer is nu teller DM451 + 48.
LD 217.13  ; Volgende alarm gevonden
AND 219.00  ; Alarm in register 6 zoeken
+BC(406) RDTELLER #97 RDALNMR  ; REG. DISPLAY 1 T/M 16, REG. DISPLAY ALARMNUMMER BCD
; rung 81: DISPLAY / Alarm in HR07, Alarmnummer is nu teller DM451 + 64.
LD 217.13  ; Volgende alarm gevonden
AND 219.01  ; Alarm in register 7 zoeken
+BC(406) RDTELLER #113 RDALNMR  ; REG. DISPLAY 1 T/M 16, REG. DISPLAY ALARMNUMMER BCD
; rung 82: DISPLAY / Alarm in HR08, Alarmnummer is nu teller DM451 + 80.
LD 217.13  ; Volgende alarm gevonden
AND 219.02  ; Alarm in register 8 zoeken
+BC(406) RDTELLER #129 RDALNMR  ; REG. DISPLAY 1 T/M 16, REG. DISPLAY ALARMNUMMER BCD
; rung 83: SUBREind / Einde subroutine 91, Aansturing display t.b.v. alarmmeldingen.
RET(093)

### Section Subroutine_Poortjes

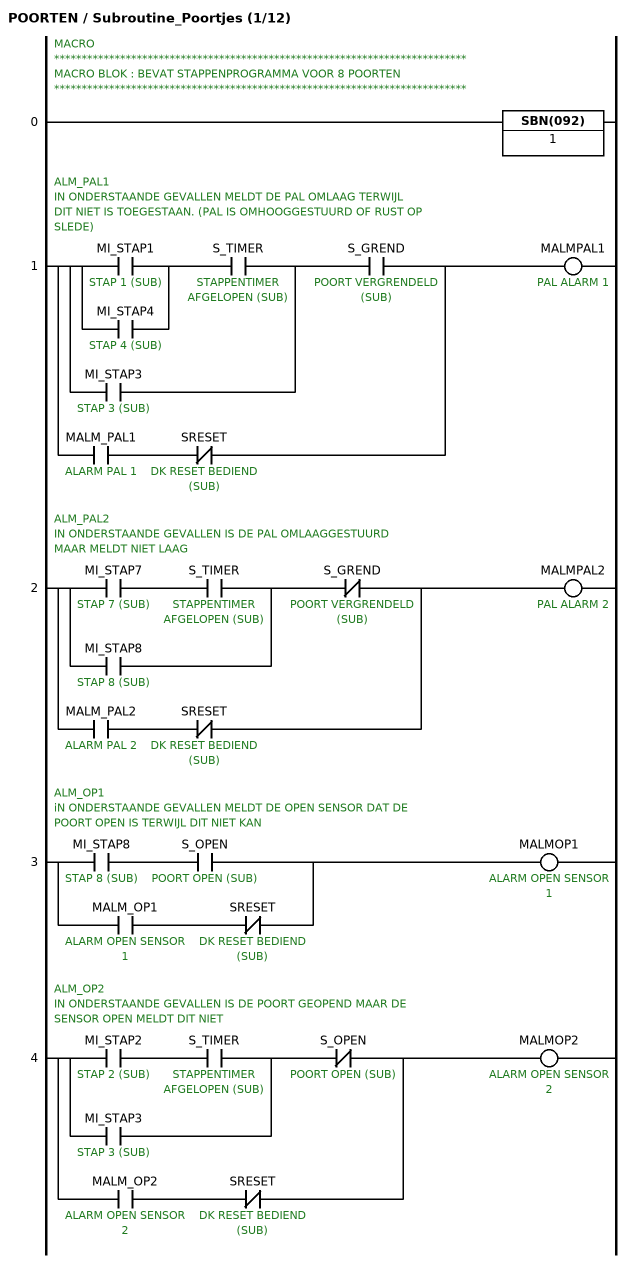
; rung 0: MACRO / *************************************************************************** / MACRO BLOK : BEVAT STAPPENPROGRAMMA VOOR 8 POORTEN / ***************************************************************************
SBN(092) 1
; rung 1: ALM_PAL1 / IN ONDERSTAANDE GEVALLEN MELDT DE PAL OMLAAG TERWIJL / DIT NIET IS TOEGESTAAN. (PAL IS OMHOOGGESTUURD OF RUST OP / SLEDE)
LD MI_STAP1  ; STAP 1 (SUB)
OR MI_STAP4  ; STAP 4 (SUB)
AND S_TIMER  ; STAPPENTIMER AFGELOPEN (SUB)
OR MI_STAP3  ; STAP 3 (SUB)
AND S_GREND  ; POORT VERGRENDELD  (SUB)
LD MALM_PAL1  ; ALARM PAL 1
ANDNOT SRESET  ; DK RESET BEDIEND (SUB)
ORLD
OUT MALMPAL1  ; PAL ALARM 1
; rung 2: ALM_PAL2 / IN ONDERSTAANDE GEVALLEN IS DE PAL OMLAAGGESTUURD / MAAR MELDT NIET LAAG
LD MI_STAP7  ; STAP 7 (SUB)
AND S_TIMER  ; STAPPENTIMER AFGELOPEN (SUB)
OR MI_STAP8  ; STAP 8 (SUB)
ANDNOT S_GREND  ; POORT VERGRENDELD  (SUB)
LD MALM_PAL2  ; ALARM PAL 2
ANDNOT SRESET  ; DK RESET BEDIEND (SUB)
ORLD
OUT MALMPAL2  ; PAL ALARM 2
; rung 3: ALM_OP1 / iN ONDERSTAANDE GEVALLEN MELDT DE OPEN SENSOR DAT DE / POORT OPEN IS TERWIJL DIT NIET KAN
LD MI_STAP8  ; STAP 8 (SUB)
AND S_OPEN  ; POORT OPEN (SUB)
LD MALM_OP1  ; ALARM OPEN SENSOR 1
ANDNOT SRESET  ; DK RESET BEDIEND (SUB)
ORLD
OUT MALMOP1  ; ALARM OPEN SENSOR 1
; rung 4: ALM_OP2 / IN ONDERSTAANDE GEVALLEN IS DE POORT GEOPEND MAAR DE / SENSOR OPEN MELDT DIT NIET
LD MI_STAP2  ; STAP 2 (SUB)
AND S_TIMER  ; STAPPENTIMER AFGELOPEN (SUB)
OR MI_STAP3  ; STAP 3 (SUB)
ANDNOT S_OPEN  ; POORT OPEN (SUB)
LD MALM_OP2  ; ALARM OPEN SENSOR 2
ANDNOT SRESET  ; DK RESET BEDIEND (SUB)
ORLD
OUT MALMOP2  ; ALARM OPEN SENSOR 2

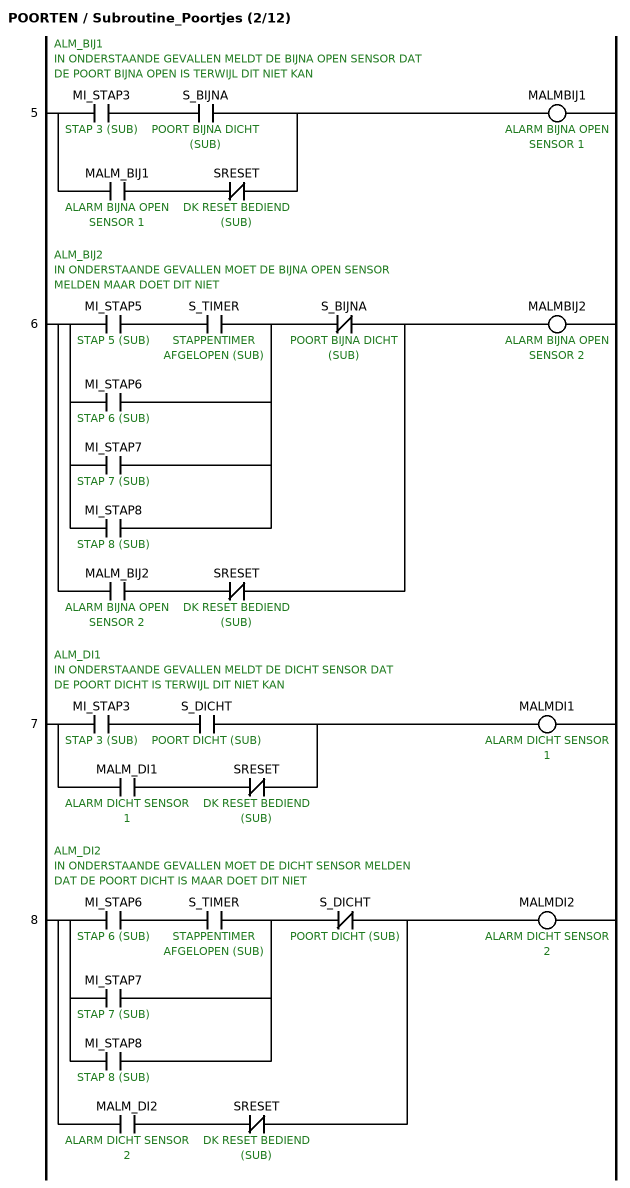
; rung 5: ALM_BIJ1 / IN ONDERSTAANDE GEVALLEN MELDT DE BIJNA OPEN SENSOR DAT / DE POORT BIJNA OPEN IS TERWIJL DIT NIET KAN
LD MI_STAP3  ; STAP 3 (SUB)
AND S_BIJNA  ; POORT BIJNA DICHT (SUB)
LD MALM_BIJ1  ; ALARM BIJNA OPEN SENSOR 1
ANDNOT SRESET  ; DK RESET BEDIEND (SUB)
ORLD
OUT MALMBIJ1  ; ALARM BIJNA OPEN SENSOR 1
; rung 6: ALM_BIJ2 / IN ONDERSTAANDE GEVALLEN MOET DE BIJNA OPEN SENSOR / MELDEN MAAR DOET DIT NIET
LD MI_STAP5  ; STAP 5 (SUB)
AND S_TIMER  ; STAPPENTIMER AFGELOPEN (SUB)
OR MI_STAP6  ; STAP 6 (SUB)
OR MI_STAP7  ; STAP 7 (SUB)
OR MI_STAP8  ; STAP 8 (SUB)
ANDNOT S_BIJNA  ; POORT BIJNA DICHT (SUB)
LD MALM_BIJ2  ; ALARM BIJNA OPEN SENSOR 2
ANDNOT SRESET  ; DK RESET BEDIEND (SUB)
ORLD
OUT MALMBIJ2  ; ALARM BIJNA OPEN SENSOR 2
; rung 7: ALM_DI1 / IN ONDERSTAANDE GEVALLEN MELDT DE DICHT SENSOR DAT / DE POORT DICHT IS TERWIJL DIT NIET KAN
LD MI_STAP3  ; STAP 3 (SUB)
AND S_DICHT  ; POORT DICHT (SUB)
LD MALM_DI1  ; ALARM DICHT SENSOR 1
ANDNOT SRESET  ; DK RESET BEDIEND (SUB)
ORLD
OUT MALMDI1  ; ALARM DICHT SENSOR 1
; rung 8: ALM_DI2 / IN ONDERSTAANDE GEVALLEN MOET DE DICHT SENSOR MELDEN / DAT DE POORT DICHT IS MAAR DOET DIT NIET
LD MI_STAP6  ; STAP 6 (SUB)
AND S_TIMER  ; STAPPENTIMER AFGELOPEN (SUB)
OR MI_STAP7  ; STAP 7 (SUB)
OR MI_STAP8  ; STAP 8 (SUB)
ANDNOT S_DICHT  ; POORT DICHT (SUB)
LD MALM_DI2  ; ALARM DICHT SENSOR 2
ANDNOT SRESET  ; DK RESET BEDIEND (SUB)
ORLD
OUT MALMDI2  ; ALARM DICHT SENSOR 2

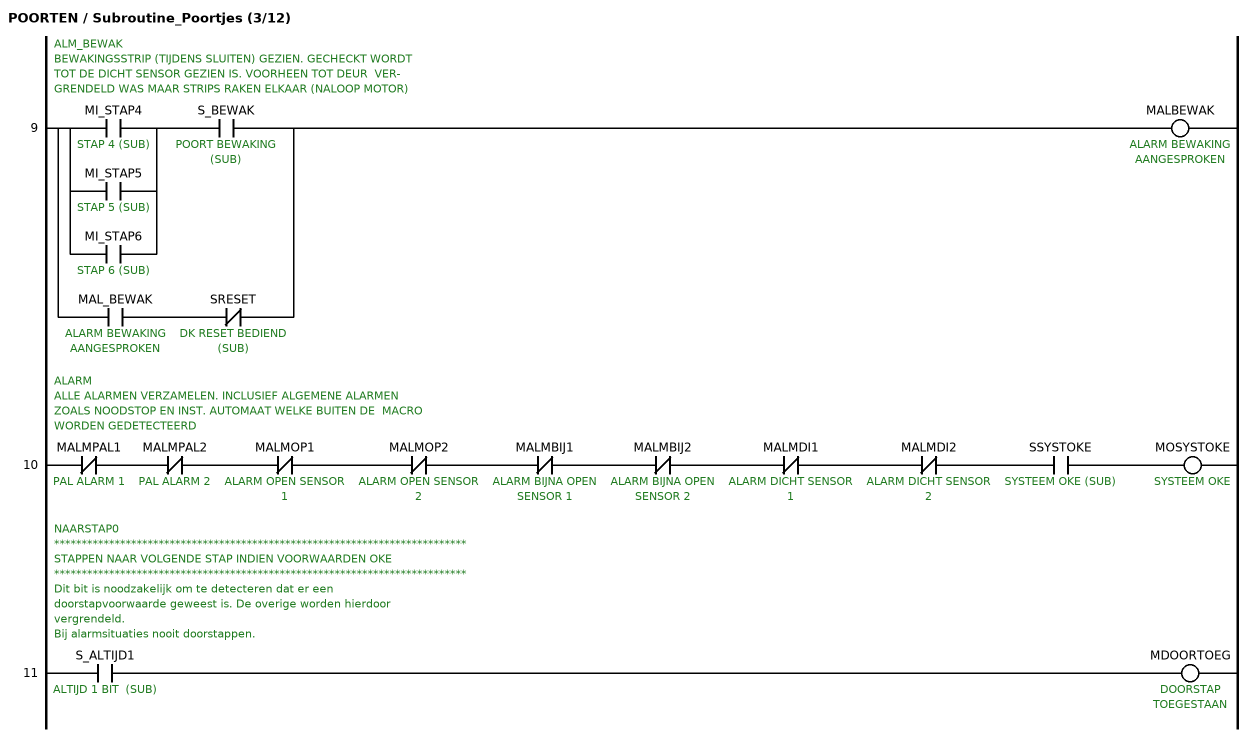
; rung 9: ALM_BEWAK / BEWAKINGSSTRIP (TIJDENS SLUITEN) GEZIEN. GECHECKT WORDT / TOT DE DICHT SENSOR GEZIEN IS. VOORHEEN TOT DEUR  VER- / GRENDELD WAS MAAR STRIPS RAKEN ELKAAR (NALOOP MOTOR)
LD MI_STAP4  ; STAP 4 (SUB)
OR MI_STAP5  ; STAP 5 (SUB)
OR MI_STAP6  ; STAP 6 (SUB)
AND S_BEWAK  ; POORT BEWAKING  (SUB)
LD MAL_BEWAK  ; ALARM BEWAKING AANGESPROKEN
ANDNOT SRESET  ; DK RESET BEDIEND (SUB)
ORLD
OUT MALBEWAK  ; ALARM BEWAKING AANGESPROKEN
; rung 10: ALARM / ALLE ALARMEN VERZAMELEN. INCLUSIEF ALGEMENE ALARMEN / ZOALS NOODSTOP EN INST. AUTOMAAT WELKE BUITEN DE  MACRO / WORDEN GEDETECTEERD
LDNOT MALMPAL1  ; PAL ALARM 1
ANDNOT MALMPAL2  ; PAL ALARM 2
ANDNOT MALMOP1  ; ALARM OPEN SENSOR 1
ANDNOT MALMOP2  ; ALARM OPEN SENSOR 2
ANDNOT MALMBIJ1  ; ALARM BIJNA OPEN SENSOR 1
ANDNOT MALMBIJ2  ; ALARM BIJNA OPEN SENSOR 2
ANDNOT MALMDI1  ; ALARM DICHT SENSOR 1
ANDNOT MALMDI2  ; ALARM DICHT SENSOR 2
AND SSYSTOKE  ; SYSTEEM OKE (SUB)
OUT MOSYSTOKE  ; SYSTEEM OKE
; rung 11: NAARSTAP0 / *************************************************************************** / STAPPEN NAAR VOLGENDE STAP INDIEN VOORWAARDEN OKE / *************************************************************************** / Dit bit is noodzakelijk om te detecteren dat er een / doorstapvoorwaarde geweest is. De overige worden hierdoor / vergrendeld. / Bij alarmsituaties nooit doorstappen.
LD S_ALTIJD1  ; ALTIJD 1 BIT  (SUB)
OUT MDOORTOEG  ; DOORSTAP TOEGESTAAN

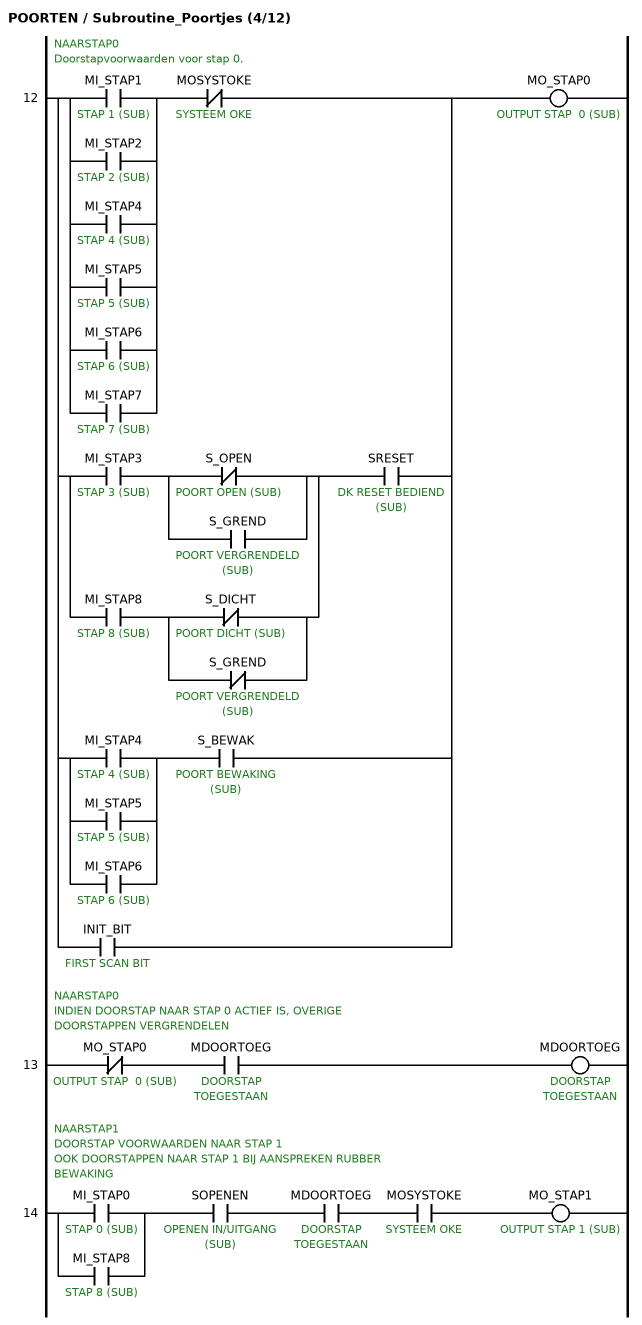
; rung 12: NAARSTAP0 / Doorstapvoorwaarden voor stap 0.
LD MI_STAP1  ; STAP 1 (SUB)
OR MI_STAP2  ; STAP 2 (SUB)
OR MI_STAP4  ; STAP 4 (SUB)
OR MI_STAP5  ; STAP 5 (SUB)
OR MI_STAP6  ; STAP 6 (SUB)
OR MI_STAP7  ; STAP 7 (SUB)
ANDNOT MOSYSTOKE  ; SYSTEEM OKE
LD MI_STAP3  ; STAP 3 (SUB)
LDNOT S_OPEN  ; POORT OPEN (SUB)
OR S_GREND  ; POORT VERGRENDELD  (SUB)
ANDLD
LD MI_STAP8  ; STAP 8 (SUB)
LDNOT S_DICHT  ; POORT DICHT (SUB)
ORNOT S_GREND  ; POORT VERGRENDELD  (SUB)
ANDLD
ORLD
AND SRESET  ; DK RESET BEDIEND (SUB)
ORLD
LD MI_STAP4  ; STAP 4 (SUB)
OR MI_STAP5  ; STAP 5 (SUB)
OR MI_STAP6  ; STAP 6 (SUB)
AND S_BEWAK  ; POORT BEWAKING  (SUB)
ORLD
OR INIT_BIT  ; FIRST SCAN BIT
OUT MO_STAP0  ; OUTPUT STAP  0 (SUB)
; rung 13: NAARSTAP0 / INDIEN DOORSTAP NAAR STAP 0 ACTIEF IS, OVERIGE / DOORSTAPPEN VERGRENDELEN
LDNOT MO_STAP0  ; OUTPUT STAP  0 (SUB)
AND MDOORTOEG  ; DOORSTAP TOEGESTAAN
OUT MDOORTOEG  ; DOORSTAP TOEGESTAAN
; rung 14: NAARSTAP1 / DOORSTAP VOORWAARDEN NAAR STAP 1 / OOK DOORSTAPPEN NAAR STAP 1 BIJ AANSPREKEN RUBBER / BEWAKING
LD MI_STAP0  ; STAP 0 (SUB)
OR MI_STAP8  ; STAP 8 (SUB)
AND SOPENEN  ; OPENEN IN/UITGANG (SUB)
AND MDOORTOEG  ; DOORSTAP TOEGESTAAN
AND MOSYSTOKE  ; SYSTEEM OKE
OUT MO_STAP1  ; OUTPUT STAP 1 (SUB)

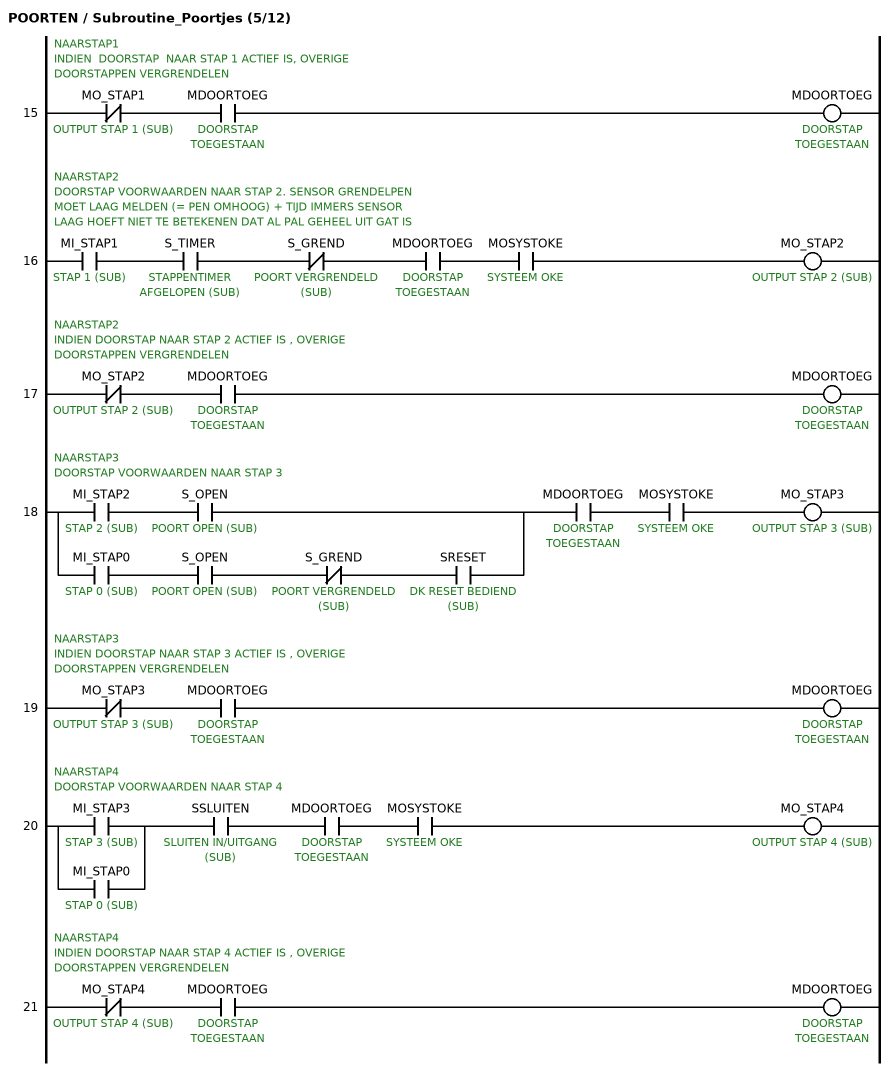
; rung 15: NAARSTAP1 / INDIEN  DOORSTAP  NAAR STAP 1 ACTIEF IS, OVERIGE / DOORSTAPPEN VERGRENDELEN
LDNOT MO_STAP1  ; OUTPUT STAP 1 (SUB)
AND MDOORTOEG  ; DOORSTAP TOEGESTAAN
OUT MDOORTOEG  ; DOORSTAP TOEGESTAAN
; rung 16: NAARSTAP2 / DOORSTAP VOORWAARDEN NAAR STAP 2. SENSOR GRENDELPEN / MOET LAAG MELDEN (= PEN OMHOOG) + TIJD IMMERS SENSOR / LAAG HOEFT NIET TE BETEKENEN DAT AL PAL GEHEEL UIT GAT IS
LD MI_STAP1  ; STAP 1 (SUB)
AND S_TIMER  ; STAPPENTIMER AFGELOPEN (SUB)
ANDNOT S_GREND  ; POORT VERGRENDELD  (SUB)
AND MDOORTOEG  ; DOORSTAP TOEGESTAAN
AND MOSYSTOKE  ; SYSTEEM OKE
OUT MO_STAP2  ; OUTPUT STAP 2 (SUB)
; rung 17: NAARSTAP2 / INDIEN DOORSTAP NAAR STAP 2 ACTIEF IS , OVERIGE / DOORSTAPPEN VERGRENDELEN
LDNOT MO_STAP2  ; OUTPUT STAP 2 (SUB)
AND MDOORTOEG  ; DOORSTAP TOEGESTAAN
OUT MDOORTOEG  ; DOORSTAP TOEGESTAAN
; rung 18: NAARSTAP3 / DOORSTAP VOORWAARDEN NAAR STAP 3
LD MI_STAP2  ; STAP 2 (SUB)
AND S_OPEN  ; POORT OPEN (SUB)
LD MI_STAP0  ; STAP 0 (SUB)
AND S_OPEN  ; POORT OPEN (SUB)
ANDNOT S_GREND  ; POORT VERGRENDELD  (SUB)
AND SRESET  ; DK RESET BEDIEND (SUB)
ORLD
AND MDOORTOEG  ; DOORSTAP TOEGESTAAN
AND MOSYSTOKE  ; SYSTEEM OKE
OUT MO_STAP3  ; OUTPUT STAP 3 (SUB)
; rung 19: NAARSTAP3 / INDIEN DOORSTAP NAAR STAP 3 ACTIEF IS , OVERIGE / DOORSTAPPEN VERGRENDELEN
LDNOT MO_STAP3  ; OUTPUT STAP 3 (SUB)
AND MDOORTOEG  ; DOORSTAP TOEGESTAAN
OUT MDOORTOEG  ; DOORSTAP TOEGESTAAN
; rung 20: NAARSTAP4 / DOORSTAP VOORWAARDEN NAAR STAP 4
LD MI_STAP3  ; STAP 3 (SUB)
OR MI_STAP0  ; STAP 0 (SUB)
AND SSLUITEN  ; SLUITEN IN/UITGANG (SUB)
AND MDOORTOEG  ; DOORSTAP TOEGESTAAN
AND MOSYSTOKE  ; SYSTEEM OKE
OUT MO_STAP4  ; OUTPUT STAP 4 (SUB)
; rung 21: NAARSTAP4 / INDIEN DOORSTAP NAAR STAP 4 ACTIEF IS , OVERIGE / DOORSTAPPEN VERGRENDELEN
LDNOT MO_STAP4  ; OUTPUT STAP 4 (SUB)
AND MDOORTOEG  ; DOORSTAP TOEGESTAAN
OUT MDOORTOEG  ; DOORSTAP TOEGESTAAN

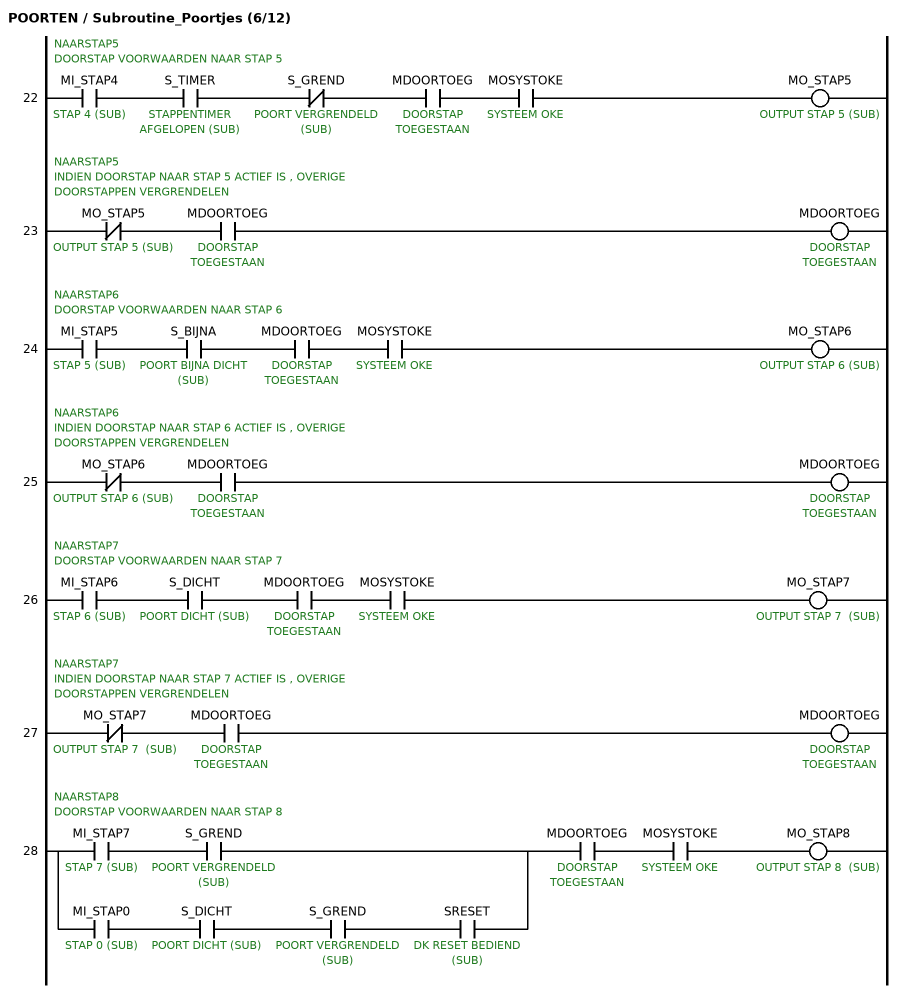
; rung 22: NAARSTAP5 / DOORSTAP VOORWAARDEN NAAR STAP 5
LD MI_STAP4  ; STAP 4 (SUB)
AND S_TIMER  ; STAPPENTIMER AFGELOPEN (SUB)
ANDNOT S_GREND  ; POORT VERGRENDELD  (SUB)
AND MDOORTOEG  ; DOORSTAP TOEGESTAAN
AND MOSYSTOKE  ; SYSTEEM OKE
OUT MO_STAP5  ; OUTPUT STAP 5 (SUB)
; rung 23: NAARSTAP5 / INDIEN DOORSTAP NAAR STAP 5 ACTIEF IS , OVERIGE / DOORSTAPPEN VERGRENDELEN
LDNOT MO_STAP5  ; OUTPUT STAP 5 (SUB)
AND MDOORTOEG  ; DOORSTAP TOEGESTAAN
OUT MDOORTOEG  ; DOORSTAP TOEGESTAAN
; rung 24: NAARSTAP6 / DOORSTAP VOORWAARDEN NAAR STAP 6
LD MI_STAP5  ; STAP 5 (SUB)
AND S_BIJNA  ; POORT BIJNA DICHT (SUB)
AND MDOORTOEG  ; DOORSTAP TOEGESTAAN
AND MOSYSTOKE  ; SYSTEEM OKE
OUT MO_STAP6  ; OUTPUT STAP 6 (SUB)
; rung 25: NAARSTAP6 / INDIEN DOORSTAP NAAR STAP 6 ACTIEF IS , OVERIGE / DOORSTAPPEN VERGRENDELEN
LDNOT MO_STAP6  ; OUTPUT STAP 6 (SUB)
AND MDOORTOEG  ; DOORSTAP TOEGESTAAN
OUT MDOORTOEG  ; DOORSTAP TOEGESTAAN
; rung 26: NAARSTAP7 / DOORSTAP VOORWAARDEN NAAR STAP 7
LD MI_STAP6  ; STAP 6 (SUB)
AND S_DICHT  ; POORT DICHT (SUB)
AND MDOORTOEG  ; DOORSTAP TOEGESTAAN
AND MOSYSTOKE  ; SYSTEEM OKE
OUT MO_STAP7  ; OUTPUT STAP 7  (SUB)
; rung 27: NAARSTAP7 / INDIEN DOORSTAP NAAR STAP 7 ACTIEF IS , OVERIGE / DOORSTAPPEN VERGRENDELEN
LDNOT MO_STAP7  ; OUTPUT STAP 7  (SUB)
AND MDOORTOEG  ; DOORSTAP TOEGESTAAN
OUT MDOORTOEG  ; DOORSTAP TOEGESTAAN
; rung 28: NAARSTAP8 / DOORSTAP VOORWAARDEN NAAR STAP 8
LD MI_STAP7  ; STAP 7 (SUB)
AND S_GREND  ; POORT VERGRENDELD  (SUB)
LD MI_STAP0  ; STAP 0 (SUB)
AND S_DICHT  ; POORT DICHT (SUB)
AND S_GREND  ; POORT VERGRENDELD  (SUB)
AND SRESET  ; DK RESET BEDIEND (SUB)
ORLD
AND MDOORTOEG  ; DOORSTAP TOEGESTAAN
AND MOSYSTOKE  ; SYSTEEM OKE
OUT MO_STAP8  ; OUTPUT STAP 8  (SUB)

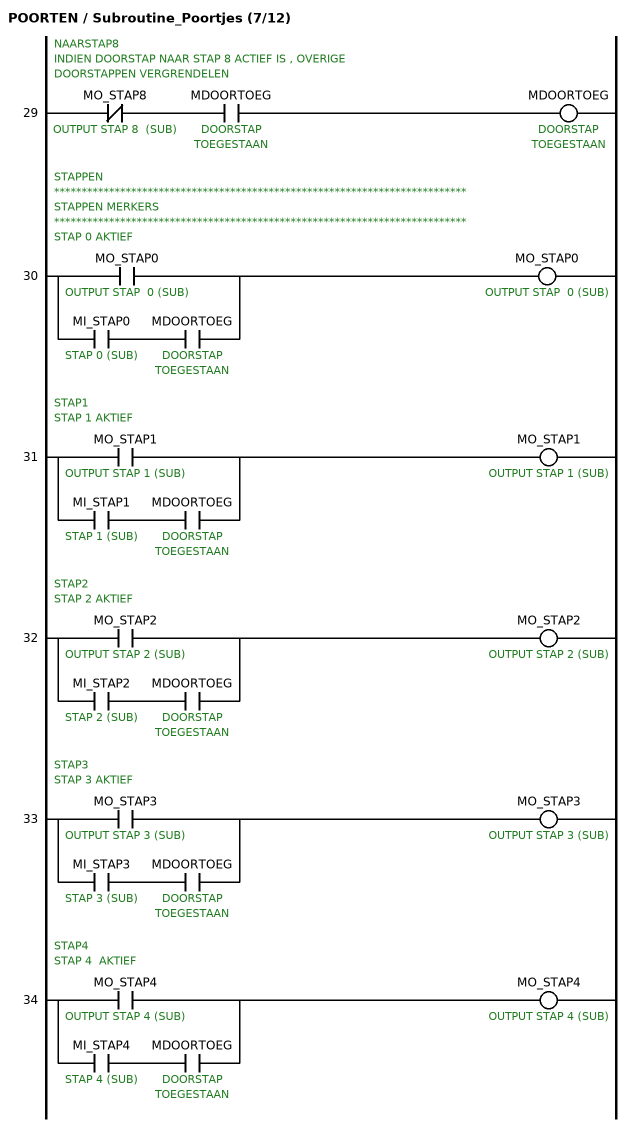
; rung 29: NAARSTAP8 / INDIEN DOORSTAP NAAR STAP 8 ACTIEF IS , OVERIGE / DOORSTAPPEN VERGRENDELEN
LDNOT MO_STAP8  ; OUTPUT STAP 8  (SUB)
AND MDOORTOEG  ; DOORSTAP TOEGESTAAN
OUT MDOORTOEG  ; DOORSTAP TOEGESTAAN
; rung 30: STAPPEN / *************************************************************************** / STAPPEN MERKERS / *************************************************************************** / STAP 0 AKTIEF
LD MO_STAP0  ; OUTPUT STAP  0 (SUB)
LD MI_STAP0  ; STAP 0 (SUB)
AND MDOORTOEG  ; DOORSTAP TOEGESTAAN
ORLD
OUT MO_STAP0  ; OUTPUT STAP  0 (SUB)
; rung 31: STAP1 / STAP 1 AKTIEF
LD MO_STAP1  ; OUTPUT STAP 1 (SUB)
LD MI_STAP1  ; STAP 1 (SUB)
AND MDOORTOEG  ; DOORSTAP TOEGESTAAN
ORLD
OUT MO_STAP1  ; OUTPUT STAP 1 (SUB)
; rung 32: STAP2 / STAP 2 AKTIEF
LD MO_STAP2  ; OUTPUT STAP 2 (SUB)
LD MI_STAP2  ; STAP 2 (SUB)
AND MDOORTOEG  ; DOORSTAP TOEGESTAAN
ORLD
OUT MO_STAP2  ; OUTPUT STAP 2 (SUB)
; rung 33: STAP3 / STAP 3 AKTIEF
LD MO_STAP3  ; OUTPUT STAP 3 (SUB)
LD MI_STAP3  ; STAP 3 (SUB)
AND MDOORTOEG  ; DOORSTAP TOEGESTAAN
ORLD
OUT MO_STAP3  ; OUTPUT STAP 3 (SUB)
; rung 34: STAP4 / STAP 4  AKTIEF
LD MO_STAP4  ; OUTPUT STAP 4 (SUB)
LD MI_STAP4  ; STAP 4 (SUB)
AND MDOORTOEG  ; DOORSTAP TOEGESTAAN
ORLD
OUT MO_STAP4  ; OUTPUT STAP 4 (SUB)

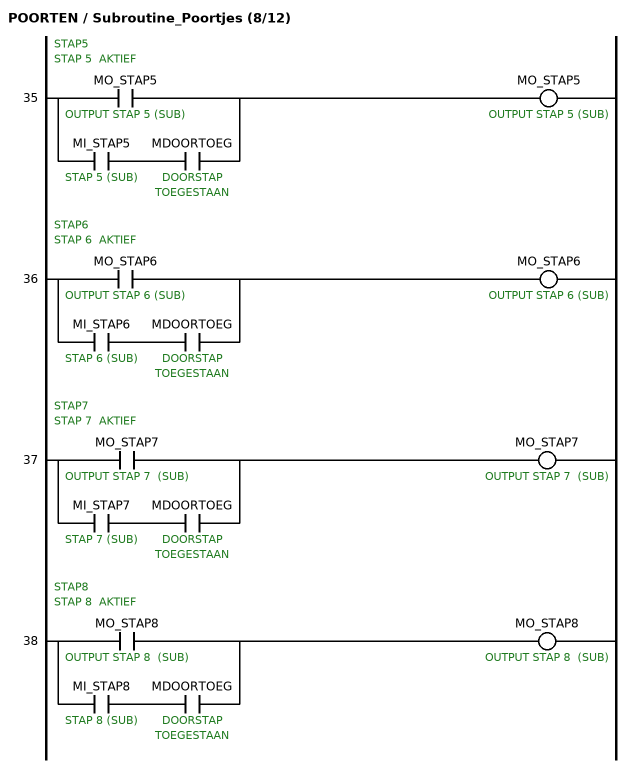
; rung 35: STAP5 / STAP 5  AKTIEF
LD MO_STAP5  ; OUTPUT STAP 5 (SUB)
LD MI_STAP5  ; STAP 5 (SUB)
AND MDOORTOEG  ; DOORSTAP TOEGESTAAN
ORLD
OUT MO_STAP5  ; OUTPUT STAP 5 (SUB)
; rung 36: STAP6 / STAP 6  AKTIEF
LD MO_STAP6  ; OUTPUT STAP 6 (SUB)
LD MI_STAP6  ; STAP 6 (SUB)
AND MDOORTOEG  ; DOORSTAP TOEGESTAAN
ORLD
OUT MO_STAP6  ; OUTPUT STAP 6 (SUB)
; rung 37: STAP7 / STAP 7  AKTIEF
LD MO_STAP7  ; OUTPUT STAP 7  (SUB)
LD MI_STAP7  ; STAP 7 (SUB)
AND MDOORTOEG  ; DOORSTAP TOEGESTAAN
ORLD
OUT MO_STAP7  ; OUTPUT STAP 7  (SUB)
; rung 38: STAP8 / STAP 8  AKTIEF
LD MO_STAP8  ; OUTPUT STAP 8  (SUB)
LD MI_STAP8  ; STAP 8 (SUB)
AND MDOORTOEG  ; DOORSTAP TOEGESTAAN
ORLD
OUT MO_STAP8  ; OUTPUT STAP 8  (SUB)

